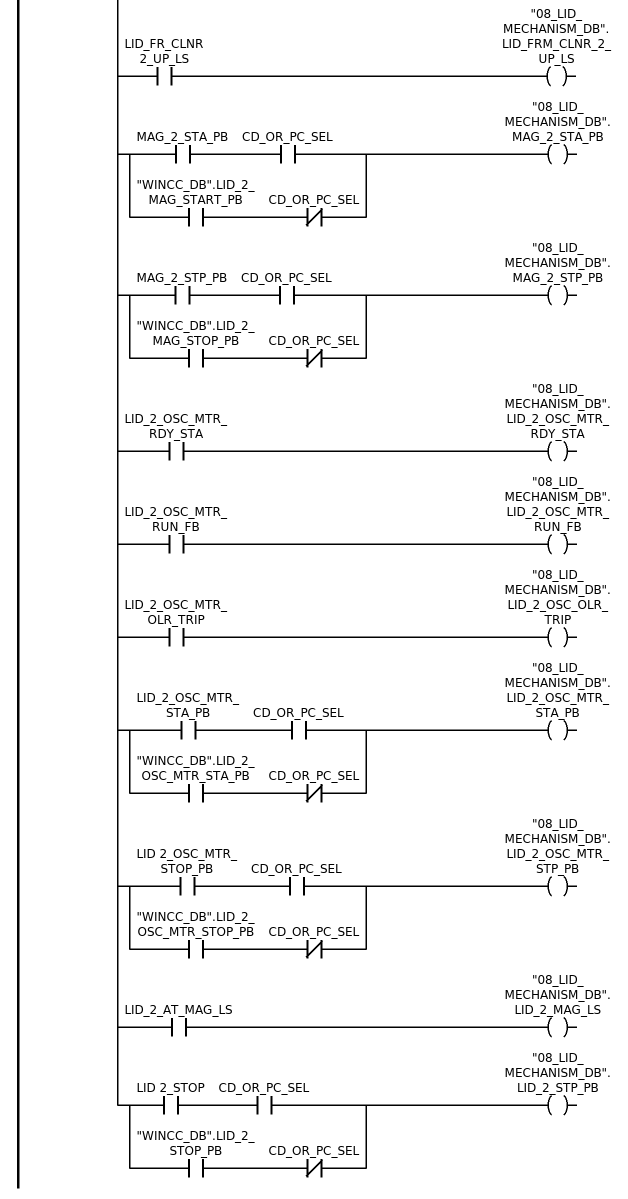
[picture p24: INPUT_MAPPING networks 7-7]
NETWORK
TITLE = LID MECHANISM 2 INPUT MAPPING
      A     "ALWAYS_ON";
      =     L 0.0;
      A     L 0.0;
      A     "LID_FR_CLN_MT_2_RDY_STA";
      =     "08_LID_MECHANISM_DB".LID_FR_CLN_MTR_2_RDY_STA;
      A     L 0.0;
      A     "LID_FR_CLN_MTR_2_RUN_FB";
      =     "08_LID_MECHANISM_DB".LID_FR_CLN_MTR_2_RUN_FB;
      A     L 0.0;
      A     "LID_FR_CLN_MTR_2_OLR";
      =     "08_LID_MECHANISM_DB".LID_FR_CLN_MTR_2_OLR_TRP;
      A     L 0.0;
      A(;
      A     "LID_FR_CL_MT_2_STA_PB";
      A     "CD_OR_PC_SEL";
      O;
      A     "WINCC_DB".LID_2_FRA_CLRMTR_STA_PB;
      AN    "CD_OR_PC_SEL";
      );
      =     "08_LID_MECHANISM_DB".LID_FR_CL_MTR_2_STA_PB;
      A     L 0.0;
      A(;
      A     "LID_FR_CLN_MTR_2_STP_PB";
      A     "CD_OR_PC_SEL";
      O;
      A     "WINCC_DB".LID_2_FRA_CLRMTR_STOP_PB;
      AN    "CD_OR_PC_SEL";
      );
      =     "08_LID_MECHANISM_DB".LID_FR_CL_MTR_2_STP_PB;
      A     L 0.0;
      A(;
      A     "LID_LIFT_2_CAR_FWD_STA";
      A     "CD_OR_PC_SEL";
      O;
      A     "WINCC_DB".LID_2_CARGE_FWD_STA_PB;
      AN    "CD_OR_PC_SEL";
      );
      =     "08_LID_MECHANISM_DB".LID_LIFT_2_CAR_FWD_STA;
      A     L 0.0;
      A(;
      A     "LID_LIFT_2_CAR_RET_STA";
      A     "CD_OR_PC_SEL";
      O;
      A     "WINCC_DB".LID_2_CARGE_REV_STA_PB;
      AN    "CD_OR_PC_SEL";
      );
      =     "08_LID_MECHANISM_DB".LID_LIFT_2_CAR_RET_STA;
      A     L 0.0;
      A(;
      A     "LID_LIFT_2_VER_DN_STA";
      A     "CD_OR_PC_SEL";
      O;
      A     "WINCC_DB".LID_2_VER_DN_STA_PB;
      AN    "CD_OR_PC_SEL";
      );
      =     "08_LID_MECHANISM_DB".LID_LIFT_2_VER_DN_STA;
      A     L 0.0;
      A(;
      A     "LID_LIFT_2_VER_UP_STA";
      A     "CD_OR_PC_SEL";
      O;
      A     "WINCC_DB".LID_2_VER_UP_STA_PB;
      AN    "CD_OR_PC_SEL";
      );
      =     "08_LID_MECHANISM_DB".LID_LIFT_2_VER_UP_STA;
      A     L 0.0;
      A(;
      A     "LID_FR_CLNR_2_DN_STA";
      A     "CD_OR_PC_SEL";
      O;
      A     "WINCC_DB".LID_2_FRA_CLR_DN_STA;
      AN    "CD_OR_PC_SEL";
      );
      =     "08_LID_MECHANISM_DB".LID_2_FRM_CLNR_DN_STA;
      A     L 0.0;
      A(;
      A     "LID_FR_CLNR_2_UP_STA";
      A     "CD_OR_PC_SEL";
      O;
      A     "WINCC_DB".LID_2_FRA_CLR_UP_STA;
      AN    "CD_OR_PC_SEL";
      );
      =     "08_LID_MECHANISM_DB".LID_2_FRM_CLNR_UP_STA;
      A     L 0.0;
      A(;
      A     "TELES_2_DOWN_STA";
      A     "CD_OR_PC_SEL";
      O;
      A     "WINCC_DB".LID_2_TELES_DN_STA;
      AN    "CD_OR_PC_SEL";
      );
      =     "08_LID_MECHANISM_DB".LID_2_TELES_DN_STA_PB;
      A     L 0.0;
      A(;
      A     "TELES_2_UP_STA";
      A     "CD_OR_PC_SEL";
      O;
      A     "WINCC_DB".LID_2_TELES_UP_STA;
      AN    "CD_OR_PC_SEL";
      );
      =     "08_LID_MECHANISM_DB".LID_2_TELES_UP_STA_PB;
      A     L 0.0;
      A     "LID_LIFT_2_CARR_FWD_LS";
      =     "08_LID_MECHANISM_DB".LID_LIFT_2_CAR_FWD_LS;
      A     L 0.0;
      A     "LID_LIFT_2_CARR_RET_LS";
      =     "08_LID_MECHANISM_DB".LID_LIFT_2_CAR_RET_LS;
      A     L 0.0;
      A     "LID_LIFT_2_VER_DN_LS";
      =     "08_LID_MECHANISM_DB".LID_LIFT_2_VER_DN_LS;
      A     L 0.0;
      A     "LID_LIFT_2_VER_UP_LS";
      =     "08_LID_MECHANISM_DB".LID_LIFT_2_VER_UP_LS;
      A     L 0.0;
      A     "TELES_2_DOWN_LS";
      =     "08_LID_MECHANISM_DB".TELE_2_DN_LS;
      A     L 0.0;
      A     "TELES_2_UP_LS";
      =     "08_LID_MECHANISM_DB".TELE_2_UP_LS;
      A     L 0.0;
      A     "LID_LIFT_2_CLN_POS_LS";
      =     "08_LID_MECHANISM_DB".LID_LIFT_2_CLN_LS;
      A     L 0.0;
      A     "LID_FR_CLNR_2_DOWN_LS";
      =     "08_LID_MECHANISM_DB".LID_FRM_CLNR_2_DN_LS;
      A     L 0.0;
      A     "LID_FR_CLNR 2_UP_LS";
      =     "08_LID_MECHANISM_DB".LID_FRM_CLNR_2_UP_LS;
      A     L 0.0;
      A(;
      A     "MAG_2_STA_PB";
      A     "CD_OR_PC_SEL";
      O;
      A     "WINCC_DB".LID_2_MAG_START_PB;
      AN    "CD_OR_PC_SEL";
      );
      =     "08_LID_MECHANISM_DB".MAG_2_STA_PB;
      A     L 0.0;
      A(;
      A     "MAG_2_STP_PB";
      A     "CD_OR_PC_SEL";
      O;
      A     "WINCC_DB".LID_2_MAG_STOP_PB;
      AN    "CD_OR_PC_SEL";
      );
      =     "08_LID_MECHANISM_DB".MAG_2_STP_PB;
      A     L 0.0;
      A     "LID_2_OSC_MTR_RDY_STA";
      =     "08_LID_MECHANISM_DB".LID_2_OSC_MTR_RDY_STA;
      A     L 0.0;
      A     "LID_2_OSC_MTR_RUN_FB";
      =     "08_LID_MECHANISM_DB".LID_2_OSC_MTR_RUN_FB;
      A     L 0.0;
      A     "LID_2_OSC_MTR_OLR_TRIP";
      =     "08_LID_MECHANISM_DB".LID_2_OSC_OLR_TRIP;
      A     L 0.0;
      A(;
      A     "LID_2_OSC_MTR_STA_PB";
      A     "CD_OR_PC_SEL";
      O;
      A     "WINCC_DB".LID_2_OSC_MTR_STA_PB;
      AN    "CD_OR_PC_SEL";
      );
      =     "08_LID_MECHANISM_DB".LID_2_OSC_MTR_STA_PB;
      A     L 0.0;
      A(;
      A     "LID 2_OSC_MTR_STOP_PB";
      A     "CD_OR_PC_SEL";
      O;
      A     "WINCC_DB".LID_2_OSC_MTR_STOP_PB;
      AN    "CD_OR_PC_SEL";
      );
      =     "08_LID_MECHANISM_DB".LID_2_OSC_MTR_STP_PB;
      A     L 0.0;
      A     "LID_2_AT_MAG_LS";
      =     "08_LID_MECHANISM_DB".LID_2_MAG_LS;
      A     L 0.0;
      A(;
      A     "LID 2_STOP";
      A     "CD_OR_PC_SEL";
      O;
      A     "WINCC_DB".LID_2_STOP_PB;
      AN    "CD_OR_PC_SEL";
      );
      =     "08_LID_MECHANISM_DB".LID_2_STP_PB;
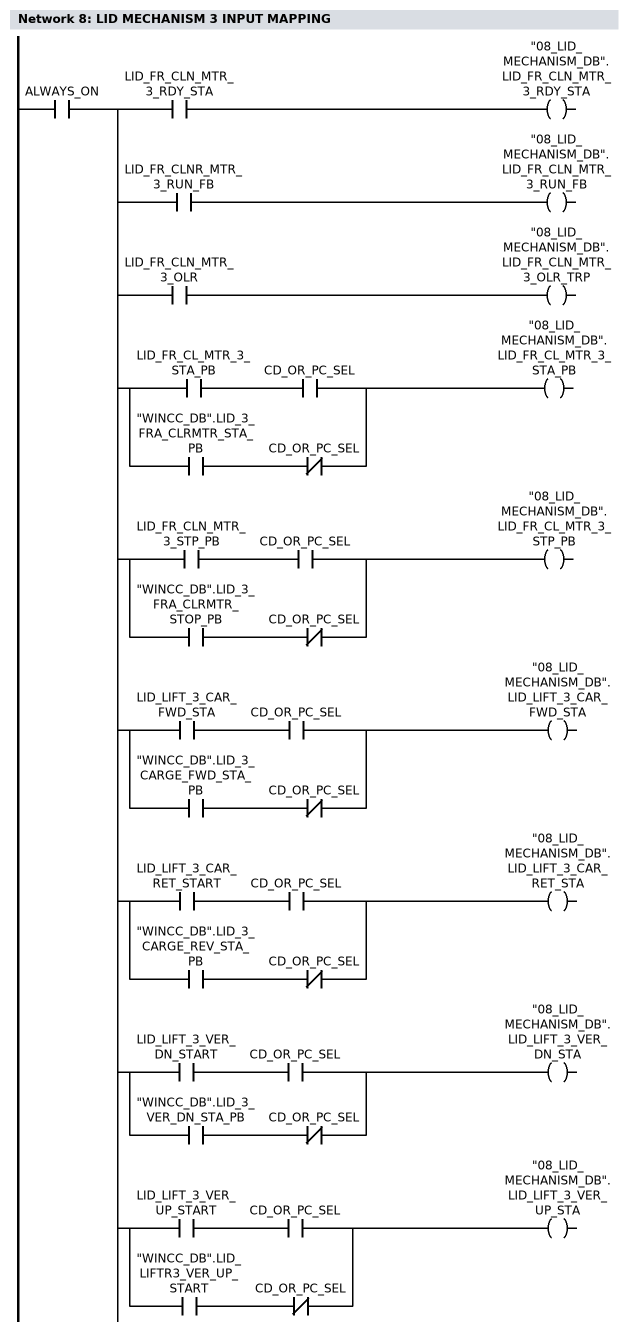
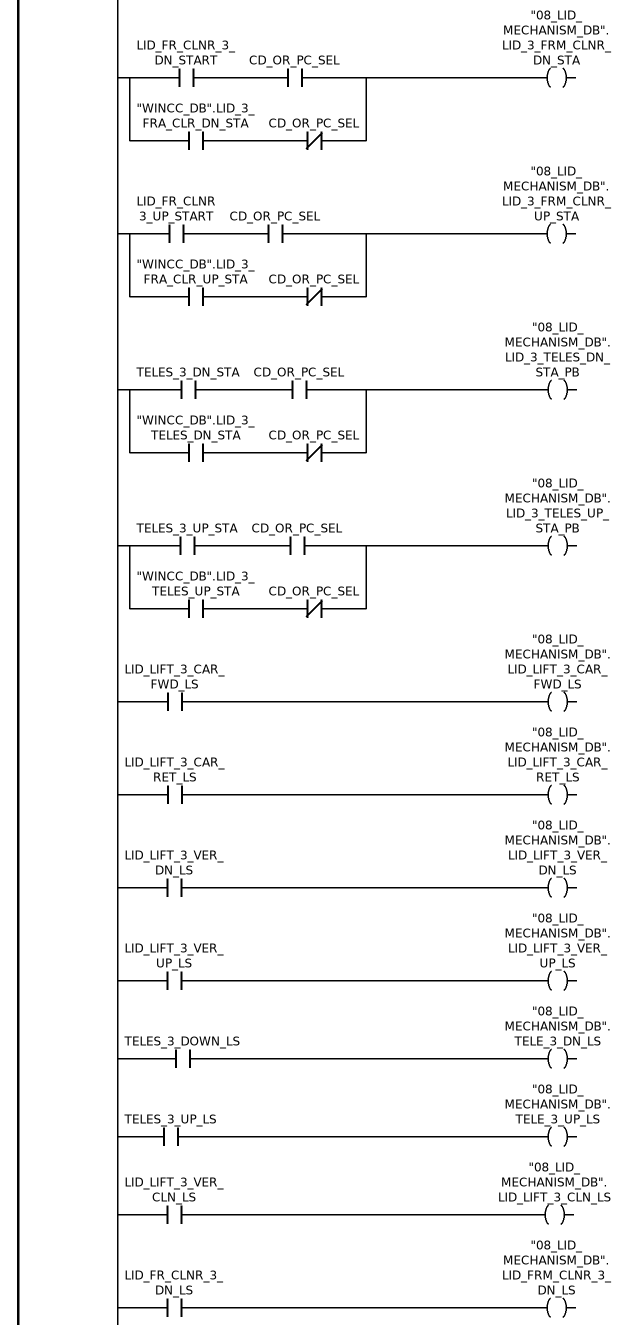
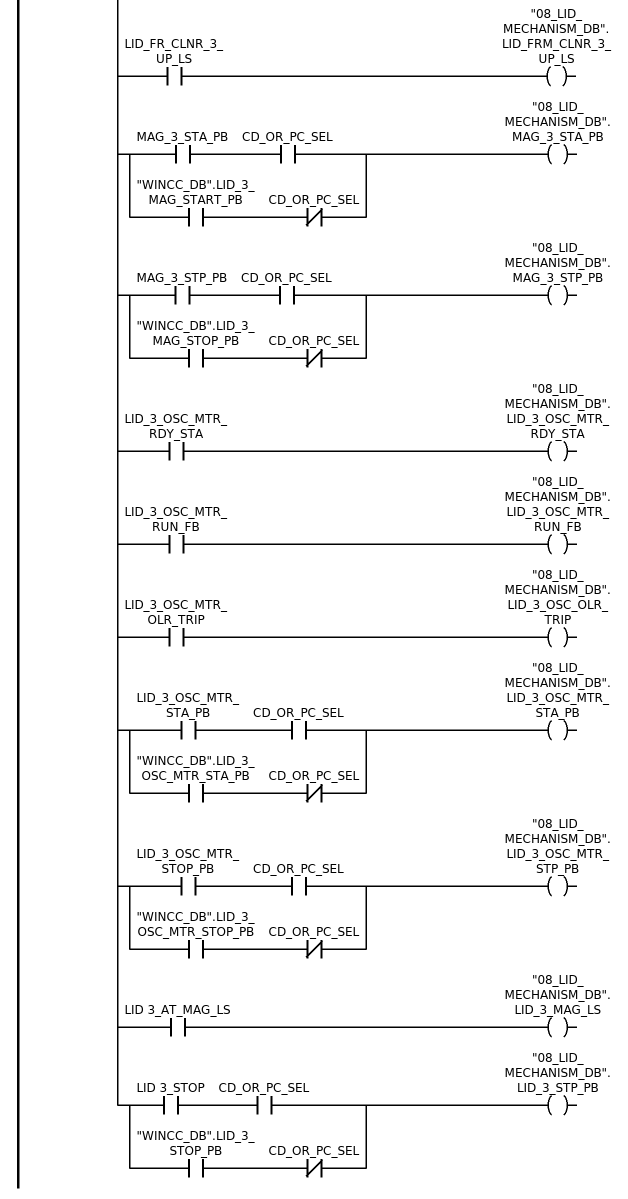
NETWORK
TITLE = LID MECHANISM 3 INPUT MAPPING
      A     "ALWAYS_ON";
      =     L 0.0;
      A     L 0.0;
      A     "LID_FR_CLN_MTR_3_RDY_STA";
      =     "08_LID_MECHANISM_DB".LID_FR_CLN_MTR_3_RDY_STA;
      A     L 0.0;
      A     "LID_FR_CLNR_MTR_3_RUN_FB";
      =     "08_LID_MECHANISM_DB".LID_FR_CLN_MTR_3_RUN_FB;
      A     L 0.0;
      A     "LID_FR_CLN_MTR_3_OLR";
      =     "08_LID_MECHANISM_DB".LID_FR_CLN_MTR_3_OLR_TRP;
      A     L 0.0;
      A(;
      A     "LID_FR_CL_MTR_3_STA_PB";
      A     "CD_OR_PC_SEL";
      O;
      A     "WINCC_DB".LID_3_FRA_CLRMTR_STA_PB;
      AN    "CD_OR_PC_SEL";
      );
      =     "08_LID_MECHANISM_DB".LID_FR_CL_MTR_3_STA_PB;
      A     L 0.0;
      A(;
      A     "LID_FR_CLN_MTR_3_STP_PB";
      A     "CD_OR_PC_SEL";
      O;
      A     "WINCC_DB".LID_3_FRA_CLRMTR_STOP_PB;
      AN    "CD_OR_PC_SEL";
      );
      =     "08_LID_MECHANISM_DB".LID_FR_CL_MTR_3_STP_PB;
      A     L 0.0;
      A(;
      A     "LID_LIFT_3_CAR_FWD_STA";
      A     "CD_OR_PC_SEL";
      O;
      A     "WINCC_DB".LID_3_CARGE_FWD_STA_PB;
      AN    "CD_OR_PC_SEL";
      );
      =     "08_LID_MECHANISM_DB".LID_LIFT_3_CAR_FWD_STA;
      A     L 0.0;
      A(;
      A     "LID_LIFT_3_CAR_RET_START";
      A     "CD_OR_PC_SEL";
      O;
      A     "WINCC_DB".LID_3_CARGE_REV_STA_PB;
      AN    "CD_OR_PC_SEL";
      );
      =     "08_LID_MECHANISM_DB".LID_LIFT_3_CAR_RET_STA;
      A     L 0.0;
      A(;
      A     "LID_LIFT_3_VER_DN_START";
      A     "CD_OR_PC_SEL";
      O;
      A     "WINCC_DB".LID_3_VER_DN_STA_PB;
      AN    "CD_OR_PC_SEL";
      );
      =     "08_LID_MECHANISM_DB".LID_LIFT_3_VER_DN_STA;
      A     L 0.0;
      A(;
      A     "LID_LIFT_3_VER_UP_START";
      A     "CD_OR_PC_SEL";
      O;
      A     "WINCC_DB".LID_LIFTR3_VER_UP_START;
      AN    "CD_OR_PC_SEL";
      );
      =     "08_LID_MECHANISM_DB".LID_LIFT_3_VER_UP_STA;
      A     L 0.0;
      A(;
      A     "LID_FR_CLNR_3_DN_START";
      A     "CD_OR_PC_SEL";
      O;
      A     "WINCC_DB".LID_3_FRA_CLR_DN_STA;
      AN    "CD_OR_PC_SEL";
      );
      =     "08_LID_MECHANISM_DB".LID_3_FRM_CLNR_DN_STA;
      A     L 0.0;
      A(;
      A     "LID_FR_CLNR 3_UP_START";
      A     "CD_OR_PC_SEL";
      O;
      A     "WINCC_DB".LID_3_FRA_CLR_UP_STA;
      AN    "CD_OR_PC_SEL";
      );
      =     "08_LID_MECHANISM_DB".LID_3_FRM_CLNR_UP_STA;
      A     L 0.0;
      A(;
      A     "TELES_3_DN_STA";
      A     "CD_OR_PC_SEL";
      O;
      A     "WINCC_DB".LID_3_TELES_DN_STA;
      AN    "CD_OR_PC_SEL";
      );
      =     "08_LID_MECHANISM_DB".LID_3_TELES_DN_STA_PB;
      A     L 0.0;
      A(;
      A     "TELES_3_UP_STA";
      A     "CD_OR_PC_SEL";
      O;
      A     "WINCC_DB".LID_3_TELES_UP_STA;
      AN    "CD_OR_PC_SEL";
      );
      =     "08_LID_MECHANISM_DB".LID_3_TELES_UP_STA_PB;
      A     L 0.0;
      A     "LID_LIFT_3_CAR_FWD_LS";
      =     "08_LID_MECHANISM_DB".LID_LIFT_3_CAR_FWD_LS;
      A     L 0.0;
      A     "LID_LIFT_3_CAR_RET_LS";
      =     "08_LID_MECHANISM_DB".LID_LIFT_3_CAR_RET_LS;
      A     L 0.0;
      A     "LID_LIFT_3_VER_DN_LS";
      =     "08_LID_MECHANISM_DB".LID_LIFT_3_VER_DN_LS;
      A     L 0.0;
      A     "LID_LIFT_3_VER_UP_LS";
      =     "08_LID_MECHANISM_DB".LID_LIFT_3_VER_UP_LS;
      A     L 0.0;
      A     "TELES_3_DOWN_LS";
      =     "08_LID_MECHANISM_DB".TELE_3_DN_LS;
      A     L 0.0;
      A     "TELES_3_UP_LS";
      =     "08_LID_MECHANISM_DB".TELE_3_UP_LS;
      A     L 0.0;
      A     "LID_LIFT_3_VER_CLN_LS";
      =     "08_LID_MECHANISM_DB".LID_LIFT_3_CLN_LS;
      A     L 0.0;
      A     "LID_FR_CLNR_3_DN_LS";
      =     "08_LID_MECHANISM_DB".LID_FRM_CLNR_3_DN_LS;
      A     L 0.0;
      A     "LID_FR_CLNR_3_UP_LS";
      =     "08_LID_MECHANISM_DB".LID_FRM_CLNR_3_UP_LS;
      A     L 0.0;
      A(;
      A     "MAG_3_STA_PB";
      A     "CD_OR_PC_SEL";
      O;
      A     "WINCC_DB".LID_3_MAG_START_PB;
      AN    "CD_OR_PC_SEL";
      );
      =     "08_LID_MECHANISM_DB".MAG_3_STA_PB;
      A     L 0.0;
      A(;
      A     "MAG_3_STP_PB";
      A     "CD_OR_PC_SEL";
      O;
      A     "WINCC_DB".LID_3_MAG_STOP_PB;
      AN    "CD_OR_PC_SEL";
      );
      =     "08_LID_MECHANISM_DB".MAG_3_STP_PB;
      A     L 0.0;
      A     "LID_3_OSC_MTR_RDY_STA";
      =     "08_LID_MECHANISM_DB".LID_3_OSC_MTR_RDY_STA;
      A     L 0.0;
      A     "LID_3_OSC_MTR_RUN_FB";
      =     "08_LID_MECHANISM_DB".LID_3_OSC_MTR_RUN_FB;
      A     L 0.0;
      A     "LID_3_OSC_MTR_OLR_TRIP";
      =     "08_LID_MECHANISM_DB".LID_3_OSC_OLR_TRIP;
      A     L 0.0;
      A(;
      A     "LID_3_OSC_MTR_STA_PB";
      A     "CD_OR_PC_SEL";
      O;
      A     "WINCC_DB".LID_3_OSC_MTR_STA_PB;
      AN    "CD_OR_PC_SEL";
      );
      =     "08_LID_MECHANISM_DB".LID_3_OSC_MTR_STA_PB;
      A     L 0.0;
      A(;
      A     "LID_3_OSC_MTR_STOP_PB";
      A     "CD_OR_PC_SEL";
      O;
      A     "WINCC_DB".LID_3_OSC_MTR_STOP_PB;
      AN    "CD_OR_PC_SEL";
      );
      =     "08_LID_MECHANISM_DB".LID_3_OSC_MTR_STP_PB;
      A     L 0.0;
      A     "LID 3_AT_MAG_LS";
      =     "08_LID_MECHANISM_DB".LID_3_MAG_LS;
      A     L 0.0;
      A(;
      A     "LID 3_STOP";
      A     "CD_OR_PC_SEL";
      O;
      A     "WINCC_DB".LID_3_STOP_PB;
      AN    "CD_OR_PC_SEL";
      );
      =     "08_LID_MECHANISM_DB".LID_3_STP_PB;
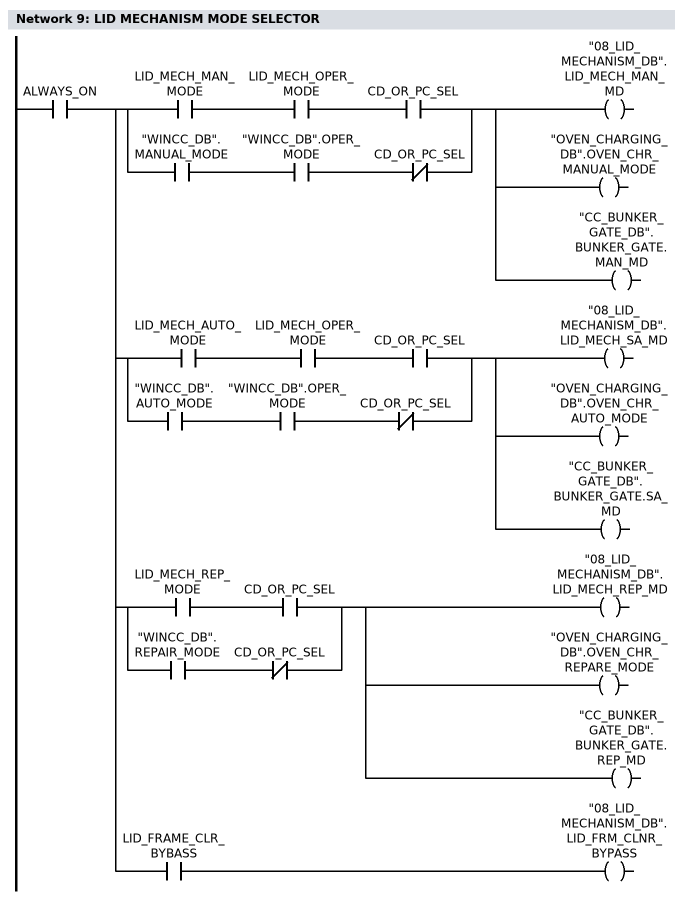
NETWORK
TITLE = LID MECHANISM MODE SELECTOR
      A     "ALWAYS_ON";
      =     L 0.0;
      A     L 0.0;
      A(;
      A     "LID_MECH_MAN_MODE";
      A     "LID_MECH_OPER_MODE";
      A     "CD_OR_PC_SEL";
      O;
      A     "WINCC_DB".MANUAL_MODE;
      A     "WINCC_DB".OPER_MODE;
      AN    "CD_OR_PC_SEL";
      );
      =     "08_LID_MECHANISM_DB".LID_MECH_MAN_MD;
      =     "OVEN_CHARGING_DB".OVEN_CHR_MANUAL_MODE;
      =     "CC_BUNKER_GATE_DB".BUNKER_GATE.MAN_MD;
      A     L 0.0;
      A(;
      A     "LID_MECH_AUTO_MODE";
      A     "LID_MECH_OPER_MODE";
      A     "CD_OR_PC_SEL";
      O;
      A     "WINCC_DB".AUTO_MODE;
      A     "WINCC_DB".OPER_MODE;
      AN    "CD_OR_PC_SEL";
      );
      =     "08_LID_MECHANISM_DB".LID_MECH_SA_MD;
      =     "OVEN_CHARGING_DB".OVEN_CHR_AUTO_MODE;
      =     "CC_BUNKER_GATE_DB".BUNKER_GATE.SA_MD;
      A     L 0.0;
      A(;
      A     "LID_MECH_REP_MODE";
      A     "CD_OR_PC_SEL";
      O;
      A     "WINCC_DB".REPAIR_MODE;
      AN    "CD_OR_PC_SEL";
      );
      =     "08_LID_MECHANISM_DB".LID_MECH_REP_MD;
      =     "OVEN_CHARGING_DB".OVEN_CHR_REPARE_MODE;
      =     "CC_BUNKER_GATE_DB".BUNKER_GATE.REP_MD;
      A     L 0.0;
      A     "LID_FRAME_CLR_BYBASS";
      =     "08_LID_MECHANISM_DB".LID_FRM_CLNR_BYPASS;
END_FUNCTION

FUNCTION "OUTPUT_MAPPING" : VOID	// FC 6
AUTHOR : Arun_Ram
VERSION : 0.1
BEGIN
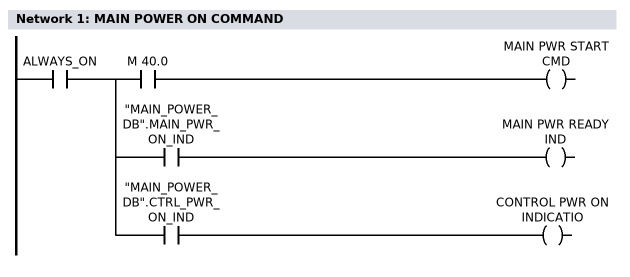
NETWORK
TITLE = MAIN POWER ON COMMAND
      A     "ALWAYS_ON";
      =     L 0.0;
      A     L 0.0;
      A     M 40.0;
      =     "MAIN PWR START CMD";
      A     L 0.0;
      A     "MAIN_POWER_DB".MAIN_PWR_ON_IND;
      =     "MAIN PWR READY IND";
      A     L 0.0;
      A     "MAIN_POWER_DB".CTRL_PWR_ON_IND;
      =     "CONTROL PWR ON INDICATIO";
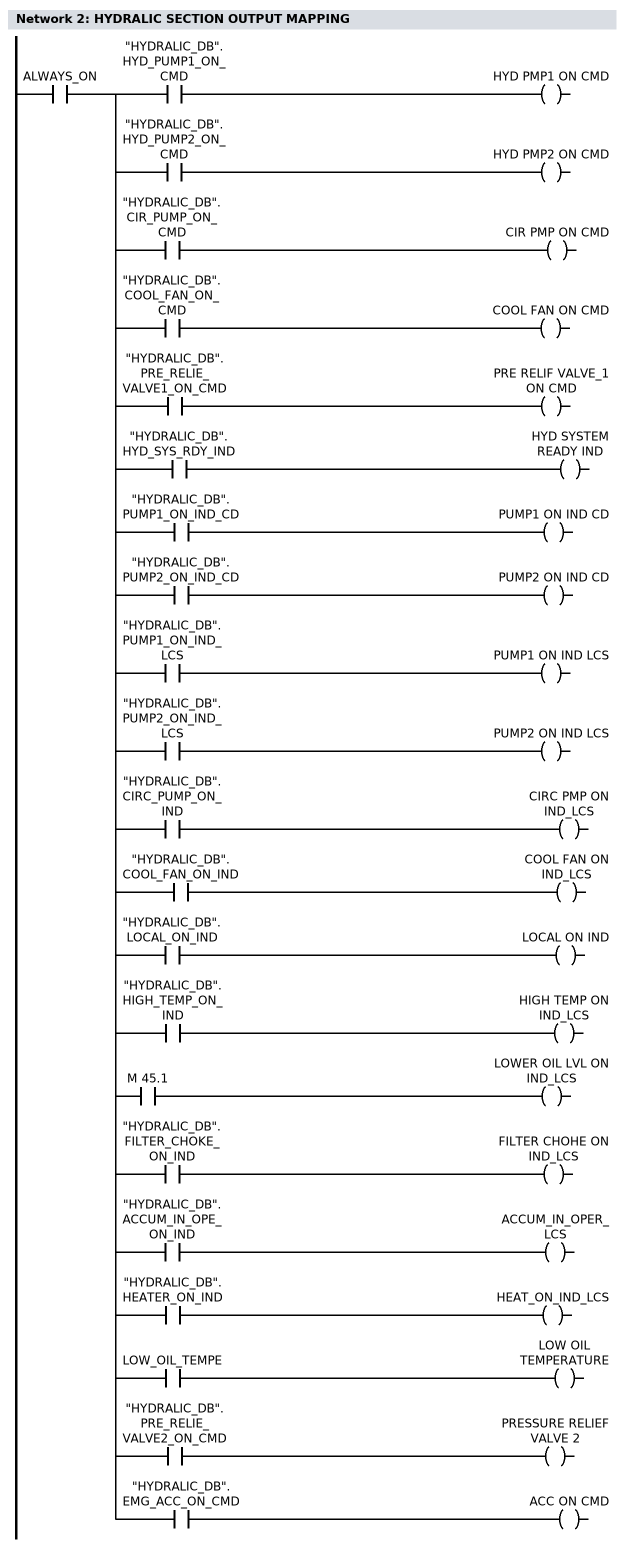
NETWORK
TITLE = HYDRALIC SECTION OUTPUT MAPPING
      A     "ALWAYS_ON";
      =     L 0.0;
      A     L 0.0;
      A     "HYDRALIC_DB".HYD_PUMP1_ON_CMD;
      =     "HYD PMP1 ON CMD";
      A     L 0.0;
      A     "HYDRALIC_DB".HYD_PUMP2_ON_CMD;
      =     "HYD PMP2 ON CMD";
      A     L 0.0;
      A     "HYDRALIC_DB".CIR_PUMP_ON_CMD;
      =     "CIR PMP ON CMD";
      A     L 0.0;
      A     "HYDRALIC_DB".COOL_FAN_ON_CMD;
      =     "COOL FAN ON CMD";
      A     L 0.0;
      A     "HYDRALIC_DB".PRE_RELIE_VALVE1_ON_CMD;
      =     "PRE RELIF VALVE_1 ON CMD";
      A     L 0.0;
      A     "HYDRALIC_DB".HYD_SYS_RDY_IND;
      =     "HYD SYSTEM READY IND";
      A     L 0.0;
      A     "HYDRALIC_DB".PUMP1_ON_IND_CD;
      =     "PUMP1 ON IND CD";
      A     L 0.0;
      A     "HYDRALIC_DB".PUMP2_ON_IND_CD;
      =     "PUMP2 ON IND CD";
      A     L 0.0;
      A     "HYDRALIC_DB".PUMP1_ON_IND_LCS;
      =     "PUMP1 ON IND LCS";
      A     L 0.0;
      A     "HYDRALIC_DB".PUMP2_ON_IND_LCS;
      =     "PUMP2 ON IND LCS";
      A     L 0.0;
      A     "HYDRALIC_DB".CIRC_PUMP_ON_IND;
      =     "CIRC PMP ON IND_LCS";
      A     L 0.0;
      A     "HYDRALIC_DB".COOL_FAN_ON_IND;
      =     "COOL FAN ON IND_LCS";
      A     L 0.0;
      A     "HYDRALIC_DB".LOCAL_ON_IND;
      =     "LOCAL ON IND";
      A     L 0.0;
      A     "HYDRALIC_DB".HIGH_TEMP_ON_IND;
      =     "HIGH TEMP ON IND_LCS";
      A     L 0.0;
      A     M 45.1;
      =     "LOWER OIL LVL ON IND_LCS";
      A     L 0.0;
      A     "HYDRALIC_DB".FILTER_CHOKE_ON_IND;
      =     "FILTER CHOHE ON IND_LCS";
      A     L 0.0;
      A     "HYDRALIC_DB".ACCUM_IN_OPE_ON_IND;
      =     "ACCUM_IN_OPER_LCS";
      A     L 0.0;
      A     "HYDRALIC_DB".HEATER_ON_IND;
      =     "HEAT_ON_IND_LCS";
      A     L 0.0;
      A     "LOW_OIL_TEMPE";
      =     "LOW OIL TEMPERATURE";
      A     L 0.0;
      A     "HYDRALIC_DB".PRE_RELIE_VALVE2_ON_CMD;
      =     "PRESSURE RELIEF VALVE 2";
      A     L 0.0;
      A     "HYDRALIC_DB".EMG_ACC_ON_CMD;
      =     "ACC ON CMD";
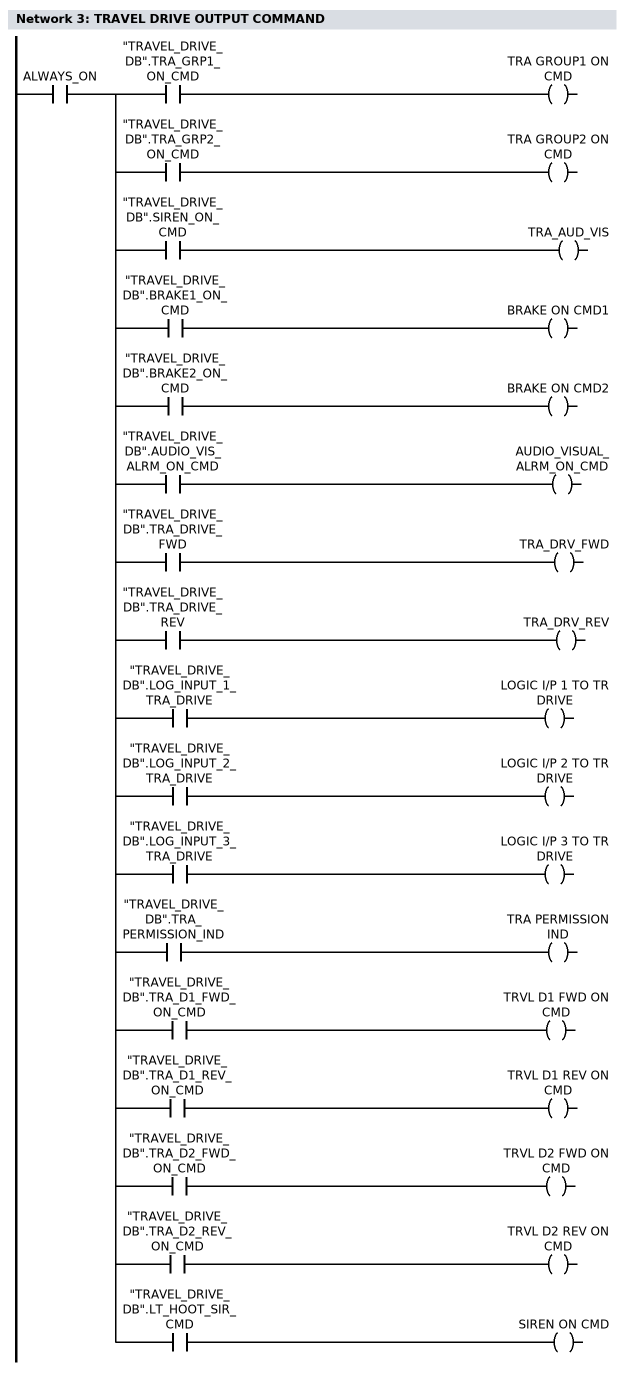
NETWORK
TITLE = TRAVEL DRIVE OUTPUT COMMAND
      A     "ALWAYS_ON";
      =     L 0.0;
      A     L 0.0;
      A     "TRAVEL_DRIVE_DB".TRA_GRP1_ON_CMD;
      =     "TRA GROUP1 ON CMD";
      A     L 0.0;
      A     "TRAVEL_DRIVE_DB".TRA_GRP2_ON_CMD;
      =     "TRA GROUP2 ON CMD";
      A     L 0.0;
      A     "TRAVEL_DRIVE_DB".SIREN_ON_CMD;
      =     "TRA_AUD_VIS";
      A     L 0.0;
      A     "TRAVEL_DRIVE_DB".BRAKE1_ON_CMD;
      =     "BRAKE ON CMD1";
      A     L 0.0;
      A     "TRAVEL_DRIVE_DB".BRAKE2_ON_CMD;
      =     "BRAKE ON CMD2";
      A     L 0.0;
      A     "TRAVEL_DRIVE_DB".AUDIO_VIS_ALRM_ON_CMD;
      =     "AUDIO_VISUAL_ALRM_ON_CMD";
      A     L 0.0;
      A     "TRAVEL_DRIVE_DB".TRA_DRIVE_FWD;
      =     "TRA_DRV_FWD";
      A     L 0.0;
      A     "TRAVEL_DRIVE_DB".TRA_DRIVE_REV;
      =     "TRA_DRV_REV";
      A     L 0.0;
      A     "TRAVEL_DRIVE_DB".LOG_INPUT_1_TRA_DRIVE;
      =     "LOGIC I/P 1 TO TR DRIVE";
      A     L 0.0;
      A     "TRAVEL_DRIVE_DB".LOG_INPUT_2_TRA_DRIVE;
      =     "LOGIC I/P 2 TO TR DRIVE";
      A     L 0.0;
      A     "TRAVEL_DRIVE_DB".LOG_INPUT_3_TRA_DRIVE;
      =     "LOGIC I/P 3 TO TR DRIVE";
      A     L 0.0;
      A     "TRAVEL_DRIVE_DB".TRA_PERMISSION_IND;
      =     "TRA PERMISSION IND";
      A     L 0.0;
      A     "TRAVEL_DRIVE_DB".TRA_D1_FWD_ON_CMD;
      =     "TRVL D1 FWD ON CMD";
      A     L 0.0;
      A     "TRAVEL_DRIVE_DB".TRA_D1_REV_ON_CMD;
      =     "TRVL D1 REV ON CMD";
      A     L 0.0;
      A     "TRAVEL_DRIVE_DB".TRA_D2_FWD_ON_CMD;
      =     "TRVL D2 FWD ON CMD";
      A     L 0.0;
      A     "TRAVEL_DRIVE_DB".TRA_D2_REV_ON_CMD;
      =     "TRVL D2 REV ON CMD";
      A     L 0.0;
      A     "TRAVEL_DRIVE_DB".LT_HOOT_SIR_CMD;
      =     "SIREN ON CMD";
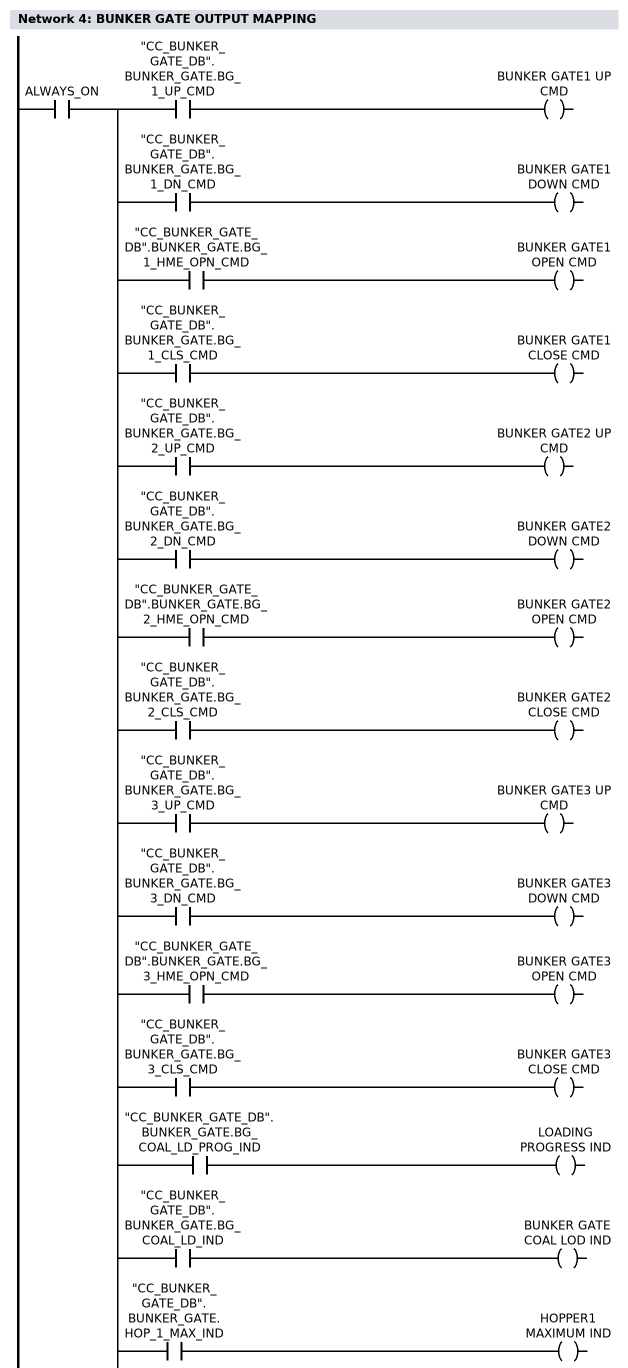
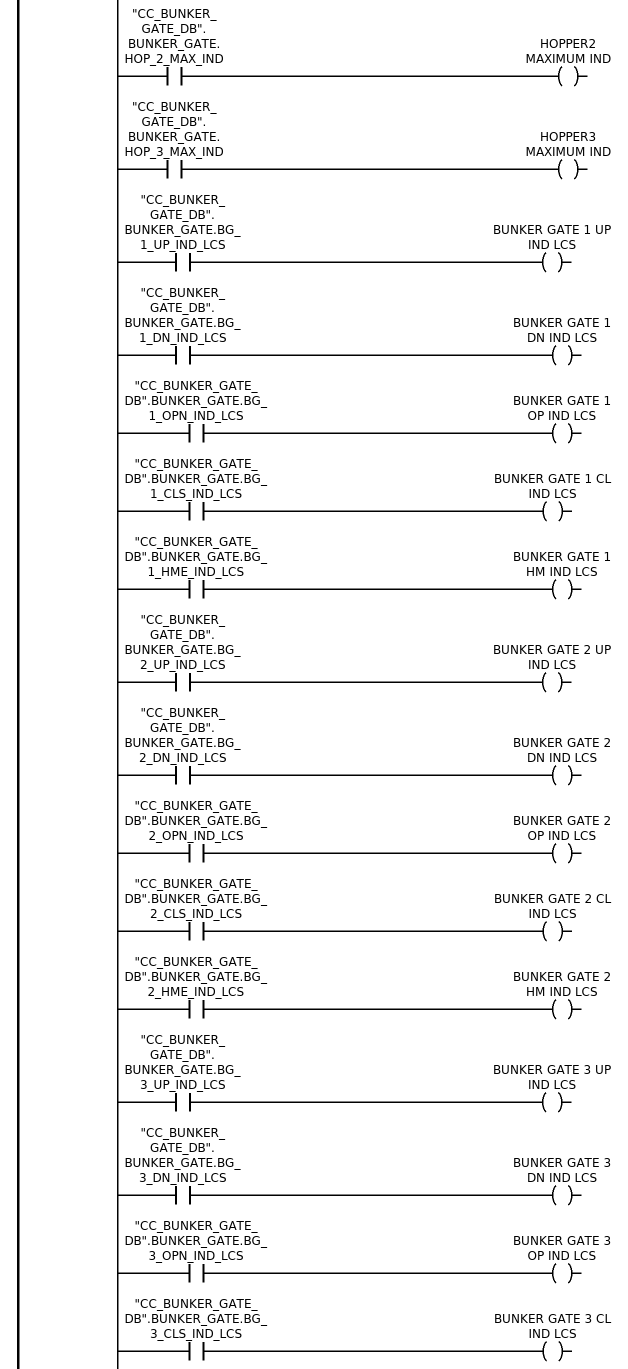
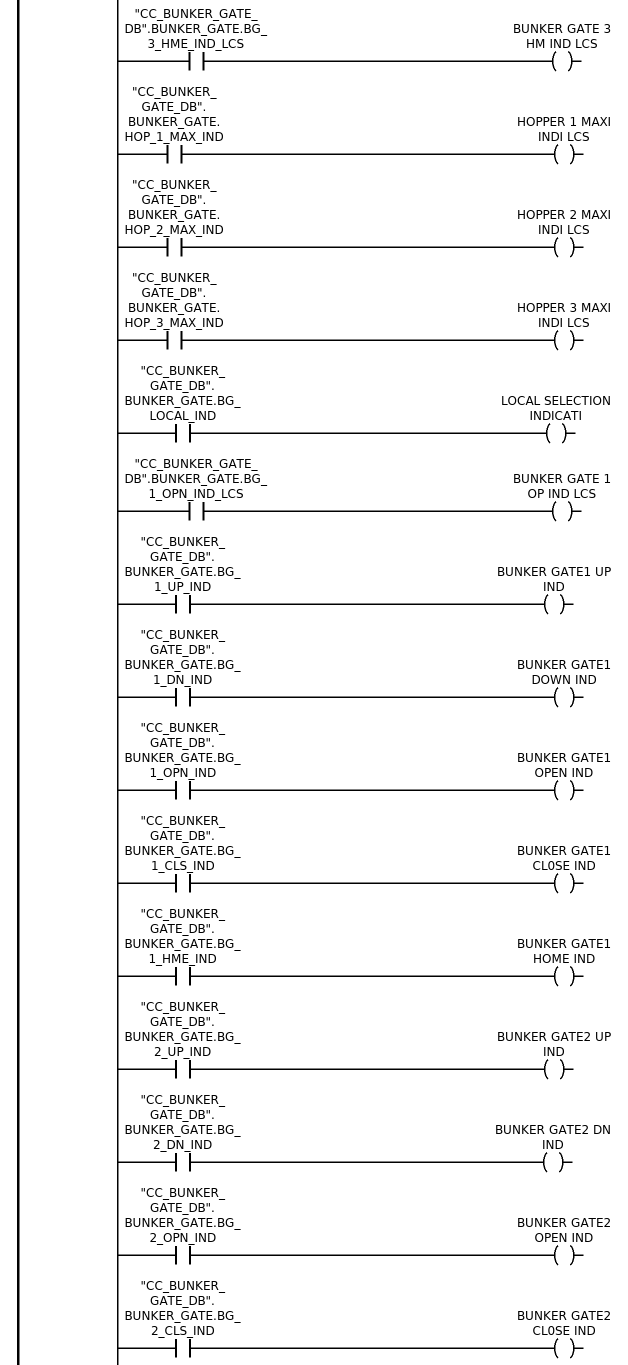
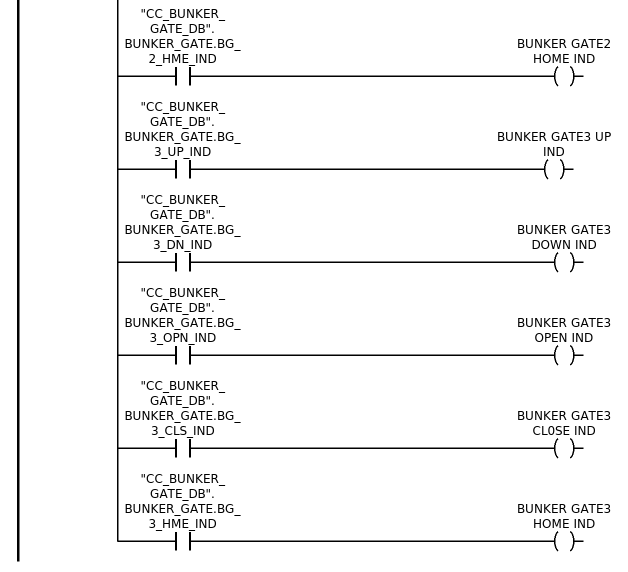
NETWORK
TITLE = BUNKER GATE OUTPUT MAPPING
      A     "ALWAYS_ON";
      =     L 0.0;
      A     L 0.0;
      A     "CC_BUNKER_GATE_DB".BUNKER_GATE.BG_1_UP_CMD;
      =     "BUNKER GATE1 UP CMD";
      A     L 0.0;
      A     "CC_BUNKER_GATE_DB".BUNKER_GATE.BG_1_DN_CMD;
      =     "BUNKER GATE1 DOWN CMD";
      A     L 0.0;
      A     "CC_BUNKER_GATE_DB".BUNKER_GATE.BG_1_HME_OPN_CMD;
      =     "BUNKER GATE1 OPEN CMD";
      A     L 0.0;
      A     "CC_BUNKER_GATE_DB".BUNKER_GATE.BG_1_CLS_CMD;
      =     "BUNKER GATE1 CLOSE CMD";
      A     L 0.0;
      A     "CC_BUNKER_GATE_DB".BUNKER_GATE.BG_2_UP_CMD;
      =     "BUNKER GATE2 UP CMD";
      A     L 0.0;
      A     "CC_BUNKER_GATE_DB".BUNKER_GATE.BG_2_DN_CMD;
      =     "BUNKER GATE2 DOWN CMD";
      A     L 0.0;
      A     "CC_BUNKER_GATE_DB".BUNKER_GATE.BG_2_HME_OPN_CMD;
      =     "BUNKER GATE2 OPEN CMD";
      A     L 0.0;
      A     "CC_BUNKER_GATE_DB".BUNKER_GATE.BG_2_CLS_CMD;
      =     "BUNKER GATE2 CLOSE CMD";
      A     L 0.0;
      A     "CC_BUNKER_GATE_DB".BUNKER_GATE.BG_3_UP_CMD;
      =     "BUNKER GATE3 UP CMD";
      A     L 0.0;
      A     "CC_BUNKER_GATE_DB".BUNKER_GATE.BG_3_DN_CMD;
      =     "BUNKER GATE3 DOWN CMD";
      A     L 0.0;
      A     "CC_BUNKER_GATE_DB".BUNKER_GATE.BG_3_HME_OPN_CMD;
      =     "BUNKER GATE3 OPEN CMD";
      A     L 0.0;
      A     "CC_BUNKER_GATE_DB".BUNKER_GATE.BG_3_CLS_CMD;
      =     "BUNKER GATE3 CLOSE CMD";
      A     L 0.0;
      A     "CC_BUNKER_GATE_DB".BUNKER_GATE.BG_COAL_LD_PROG_IND;
      =     "LOADING PROGRESS IND";
      A     L 0.0;
      A     "CC_BUNKER_GATE_DB".BUNKER_GATE.BG_COAL_LD_IND;
      =     "BUNKER GATE COAL LOD IND";
      A     L 0.0;
      A     "CC_BUNKER_GATE_DB".BUNKER_GATE.HOP_1_MAX_IND;
      =     "HOPPER1 MAXIMUM IND";
      A     L 0.0;
      A     "CC_BUNKER_GATE_DB".BUNKER_GATE.HOP_2_MAX_IND;
      =     "HOPPER2 MAXIMUM IND";
      A     L 0.0;
      A     "CC_BUNKER_GATE_DB".BUNKER_GATE.HOP_3_MAX_IND;
      =     "HOPPER3 MAXIMUM IND";
      A     L 0.0;
      A     "CC_BUNKER_GATE_DB".BUNKER_GATE.BG_1_UP_IND_LCS;
      =     "BUNKER GATE 1 UP IND LCS";
      A     L 0.0;
      A     "CC_BUNKER_GATE_DB".BUNKER_GATE.BG_1_DN_IND_LCS;
      =     "BUNKER GATE 1 DN IND LCS";
      A     L 0.0;
      A     "CC_BUNKER_GATE_DB".BUNKER_GATE.BG_1_OPN_IND_LCS;
      =     "BUNKER GATE 1 OP IND LCS";
      A     L 0.0;
      A     "CC_BUNKER_GATE_DB".BUNKER_GATE.BG_1_CLS_IND_LCS;
      =     "BUNKER GATE 1 CL IND LCS";
      A     L 0.0;
      A     "CC_BUNKER_GATE_DB".BUNKER_GATE.BG_1_HME_IND_LCS;
      =     "BUNKER GATE 1 HM IND LCS";
      A     L 0.0;
      A     "CC_BUNKER_GATE_DB".BUNKER_GATE.BG_2_UP_IND_LCS;
      =     "BUNKER GATE 2 UP IND LCS";
      A     L 0.0;
      A     "CC_BUNKER_GATE_DB".BUNKER_GATE.BG_2_DN_IND_LCS;
      =     "BUNKER GATE 2 DN IND LCS";
      A     L 0.0;
      A     "CC_BUNKER_GATE_DB".BUNKER_GATE.BG_2_OPN_IND_LCS;
      =     "BUNKER GATE 2 OP IND LCS";
      A     L 0.0;
      A     "CC_BUNKER_GATE_DB".BUNKER_GATE.BG_2_CLS_IND_LCS;
      =     "BUNKER GATE 2 CL IND LCS";
      A     L 0.0;
      A     "CC_BUNKER_GATE_DB".BUNKER_GATE.BG_2_HME_IND_LCS;
      =     "BUNKER GATE 2 HM IND LCS";
      A     L 0.0;
      A     "CC_BUNKER_GATE_DB".BUNKER_GATE.BG_3_UP_IND_LCS;
      =     "BUNKER GATE 3 UP IND LCS";
      A     L 0.0;
      A     "CC_BUNKER_GATE_DB".BUNKER_GATE.BG_3_DN_IND_LCS;
      =     "BUNKER GATE 3 DN IND LCS";
      A     L 0.0;
      A     "CC_BUNKER_GATE_DB".BUNKER_GATE.BG_3_OPN_IND_LCS;
      =     "BUNKER GATE 3 OP IND LCS";
      A     L 0.0;
      A     "CC_BUNKER_GATE_DB".BUNKER_GATE.BG_3_CLS_IND_LCS;
      =     "BUNKER GATE 3 CL IND LCS";
      A     L 0.0;
      A     "CC_BUNKER_GATE_DB".BUNKER_GATE.BG_3_HME_IND_LCS;
      =     "BUNKER GATE 3 HM IND LCS";
      A     L 0.0;
      A     "CC_BUNKER_GATE_DB".BUNKER_GATE.HOP_1_MAX_IND;
      =     "HOPPER 1 MAXI INDI LCS";
      A     L 0.0;
      A     "CC_BUNKER_GATE_DB".BUNKER_GATE.HOP_2_MAX_IND;
      =     "HOPPER 2 MAXI INDI LCS";
      A     L 0.0;
      A     "CC_BUNKER_GATE_DB".BUNKER_GATE.HOP_3_MAX_IND;
      =     "HOPPER 3 MAXI INDI LCS";
      A     L 0.0;
      A     "CC_BUNKER_GATE_DB".BUNKER_GATE.BG_LOCAL_IND;
      =     "LOCAL SELECTION INDICATI";
      A     L 0.0;
      A     "CC_BUNKER_GATE_DB".BUNKER_GATE.BG_1_OPN_IND_LCS;
      =     "BUNKER GATE 1 OP IND LCS";
      A     L 0.0;
      A     "CC_BUNKER_GATE_DB".BUNKER_GATE.BG_1_UP_IND;
      =     "BUNKER GATE1 UP IND";
      A     L 0.0;
      A     "CC_BUNKER_GATE_DB".BUNKER_GATE.BG_1_DN_IND;
      =     "BUNKER GATE1 DOWN IND";
      A     L 0.0;
      A     "CC_BUNKER_GATE_DB".BUNKER_GATE.BG_1_OPN_IND;
      =     "BUNKER GATE1 OPEN IND";
      A     L 0.0;
      A     "CC_BUNKER_GATE_DB".BUNKER_GATE.BG_1_CLS_IND;
      =     "BUNKER GATE1 CL0SE IND";
      A     L 0.0;
      A     "CC_BUNKER_GATE_DB".BUNKER_GATE.BG_1_HME_IND;
      =     "BUNKER GATE1 HOME IND";
      A     L 0.0;
      A     "CC_BUNKER_GATE_DB".BUNKER_GATE.BG_2_UP_IND;
      =     "BUNKER GATE2 UP IND";
      A     L 0.0;
      A     "CC_BUNKER_GATE_DB".BUNKER_GATE.BG_2_DN_IND;
      =     "BUNKER GATE2 DN IND";
      A     L 0.0;
      A     "CC_BUNKER_GATE_DB".BUNKER_GATE.BG_2_OPN_IND;
      =     "BUNKER GATE2 OPEN IND";
      A     L 0.0;
      A     "CC_BUNKER_GATE_DB".BUNKER_GATE.BG_2_CLS_IND;
      =     "BUNKER GATE2 CL0SE IND";
      A     L 0.0;
      A     "CC_BUNKER_GATE_DB".BUNKER_GATE.BG_2_HME_IND;
      =     "BUNKER GATE2 HOME IND";
      A     L 0.0;
      A     "CC_BUNKER_GATE_DB".BUNKER_GATE.BG_3_UP_IND;
      =     "BUNKER GATE3 UP IND";
      A     L 0.0;
      A     "CC_BUNKER_GATE_DB".BUNKER_GATE.BG_3_DN_IND;
      =     "BUNKER GATE3 DOWN IND";
      A     L 0.0;
      A     "CC_BUNKER_GATE_DB".BUNKER_GATE.BG_3_OPN_IND;
      =     "BUNKER GATE3 OPEN IND";
      A     L 0.0;
      A     "CC_BUNKER_GATE_DB".BUNKER_GATE.BG_3_CLS_IND;
      =     "BUNKER GATE3 CL0SE IND";
      A     L 0.0;
      A     "CC_BUNKER_GATE_DB".BUNKER_GATE.BG_3_HME_IND;
      =     "BUNKER GATE3 HOME IND";
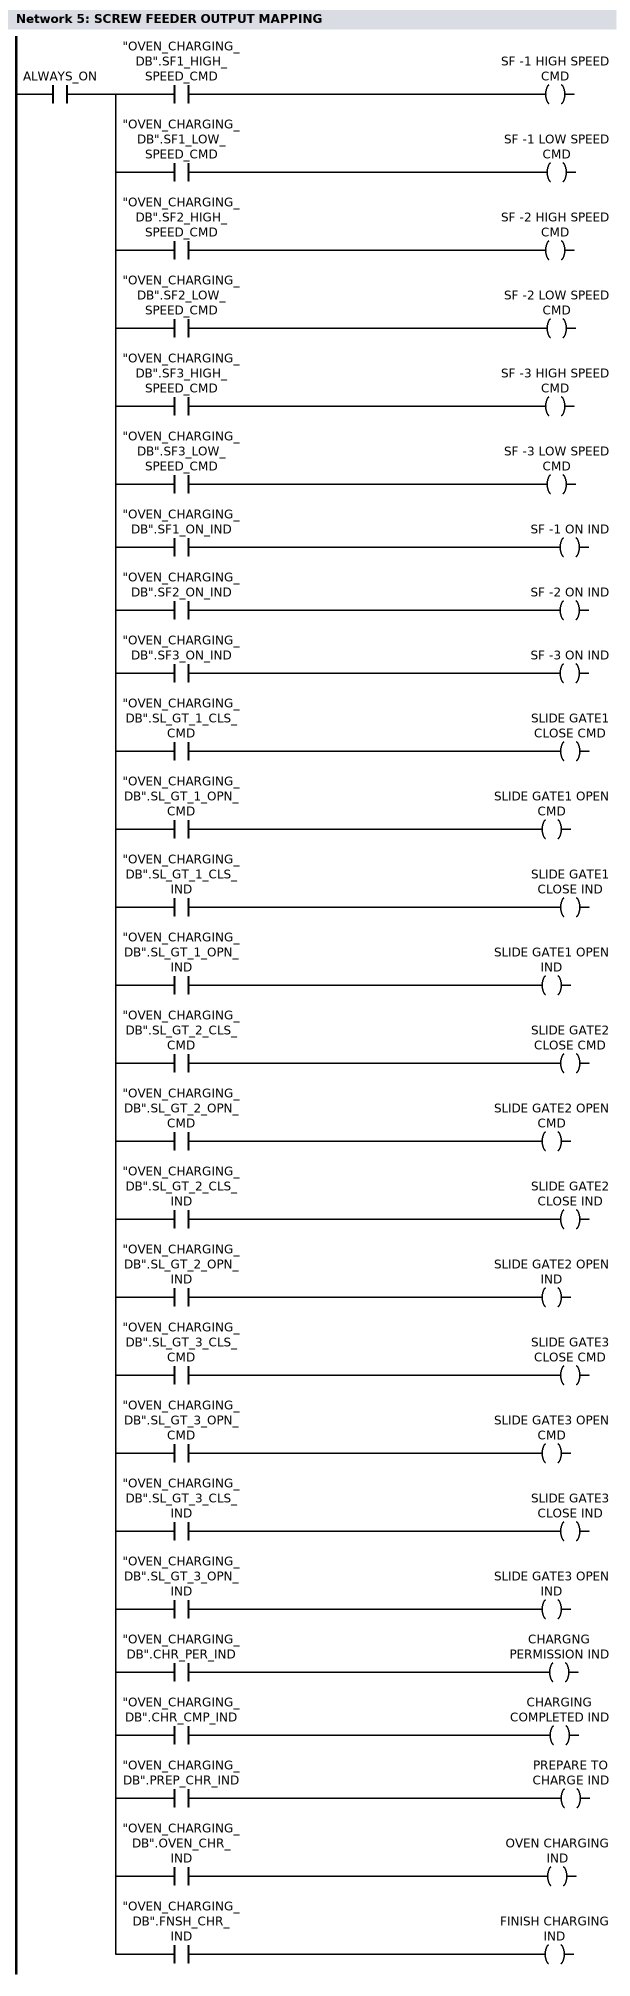
NETWORK
TITLE = SCREW FEEDER OUTPUT MAPPING
      A     "ALWAYS_ON";
      =     L 0.0;
      A     L 0.0;
      A     "OVEN_CHARGING_DB".SF1_HIGH_SPEED_CMD;
      =     "SF -1 HIGH SPEED CMD";
      A     L 0.0;
      A     "OVEN_CHARGING_DB".SF1_LOW_SPEED_CMD;
      =     "SF -1 LOW SPEED CMD";
      A     L 0.0;
      A     "OVEN_CHARGING_DB".SF2_HIGH_SPEED_CMD;
      =     "SF -2 HIGH SPEED CMD";
      A     L 0.0;
      A     "OVEN_CHARGING_DB".SF2_LOW_SPEED_CMD;
      =     "SF -2 LOW SPEED CMD";
      A     L 0.0;
      A     "OVEN_CHARGING_DB".SF3_HIGH_SPEED_CMD;
      =     "SF -3 HIGH SPEED CMD";
      A     L 0.0;
      A     "OVEN_CHARGING_DB".SF3_LOW_SPEED_CMD;
      =     "SF -3 LOW SPEED CMD";
      A     L 0.0;
      A     "OVEN_CHARGING_DB".SF1_ON_IND;
      =     "SF -1 ON IND";
      A     L 0.0;
      A     "OVEN_CHARGING_DB".SF2_ON_IND;
      =     "SF -2 ON IND";
      A     L 0.0;
      A     "OVEN_CHARGING_DB".SF3_ON_IND;
      =     "SF -3 ON IND";
      A     L 0.0;
      A     "OVEN_CHARGING_DB".SL_GT_1_CLS_CMD;
      =     "SLIDE GATE1 CLOSE CMD";
      A     L 0.0;
      A     "OVEN_CHARGING_DB".SL_GT_1_OPN_CMD;
      =     "SLIDE GATE1 OPEN CMD";
      A     L 0.0;
      A     "OVEN_CHARGING_DB".SL_GT_1_CLS_IND;
      =     "SLIDE GATE1 CLOSE IND";
      A     L 0.0;
      A     "OVEN_CHARGING_DB".SL_GT_1_OPN_IND;
      =     "SLIDE GATE1 OPEN IND";
      A     L 0.0;
      A     "OVEN_CHARGING_DB".SL_GT_2_CLS_CMD;
      =     "SLIDE GATE2 CLOSE CMD";
      A     L 0.0;
      A     "OVEN_CHARGING_DB".SL_GT_2_OPN_CMD;
      =     "SLIDE GATE2 OPEN CMD";
      A     L 0.0;
      A     "OVEN_CHARGING_DB".SL_GT_2_CLS_IND;
      =     "SLIDE GATE2 CLOSE IND";
      A     L 0.0;
      A     "OVEN_CHARGING_DB".SL_GT_2_OPN_IND;
      =     "SLIDE GATE2 OPEN IND";
      A     L 0.0;
      A     "OVEN_CHARGING_DB".SL_GT_3_CLS_CMD;
      =     "SLIDE GATE3 CLOSE CMD";
      A     L 0.0;
      A     "OVEN_CHARGING_DB".SL_GT_3_OPN_CMD;
      =     "SLIDE GATE3 OPEN CMD";
      A     L 0.0;
      A     "OVEN_CHARGING_DB".SL_GT_3_CLS_IND;
      =     "SLIDE GATE3 CLOSE IND";
      A     L 0.0;
      A     "OVEN_CHARGING_DB".SL_GT_3_OPN_IND;
      =     "SLIDE GATE3 OPEN IND";
      A     L 0.0;
      A     "OVEN_CHARGING_DB".CHR_PER_IND;
      =     "CHARGNG PERMISSION IND";
      A     L 0.0;
      A     "OVEN_CHARGING_DB".CHR_CMP_IND;
      =     "CHARGING COMPLETED IND";
      A     L 0.0;
      A     "OVEN_CHARGING_DB".PREP_CHR_IND;
      =     "PREPARE TO CHARGE IND";
      A     L 0.0;
      A     "OVEN_CHARGING_DB".OVEN_CHR_IND;
      =     "OVEN CHARGING IND";
      A     L 0.0;
      A     "OVEN_CHARGING_DB".FNSH_CHR_IND;
      =     "FINISH CHARGING IND";
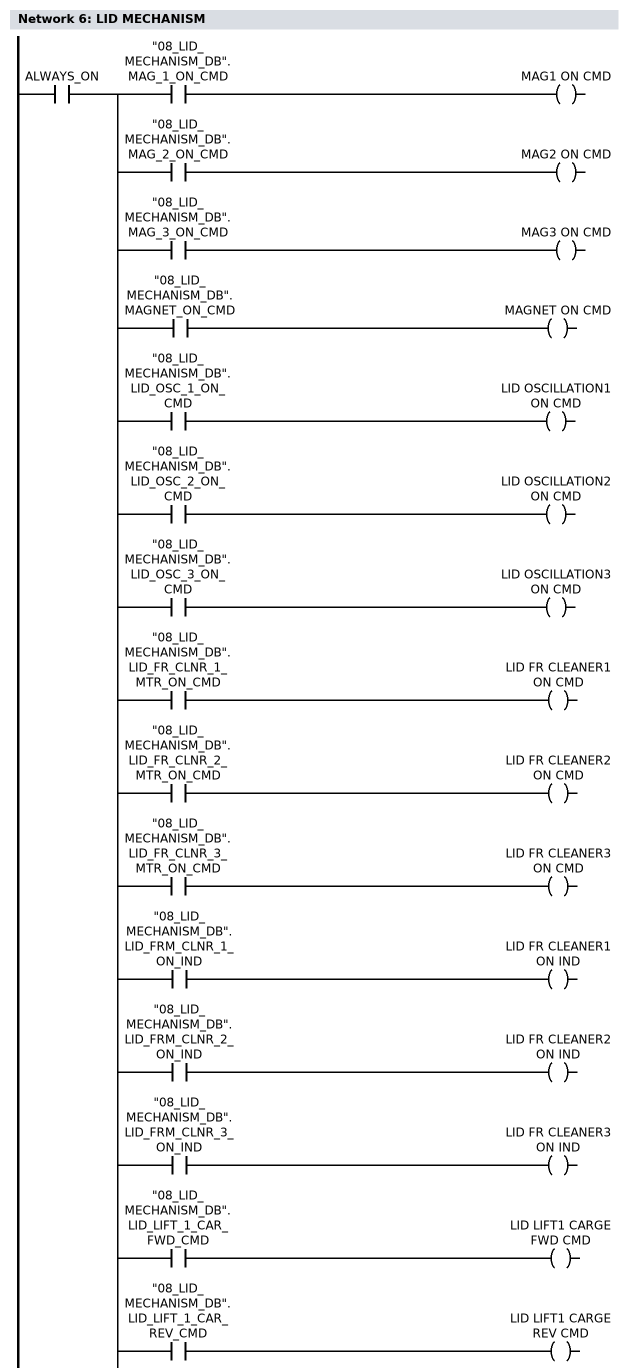
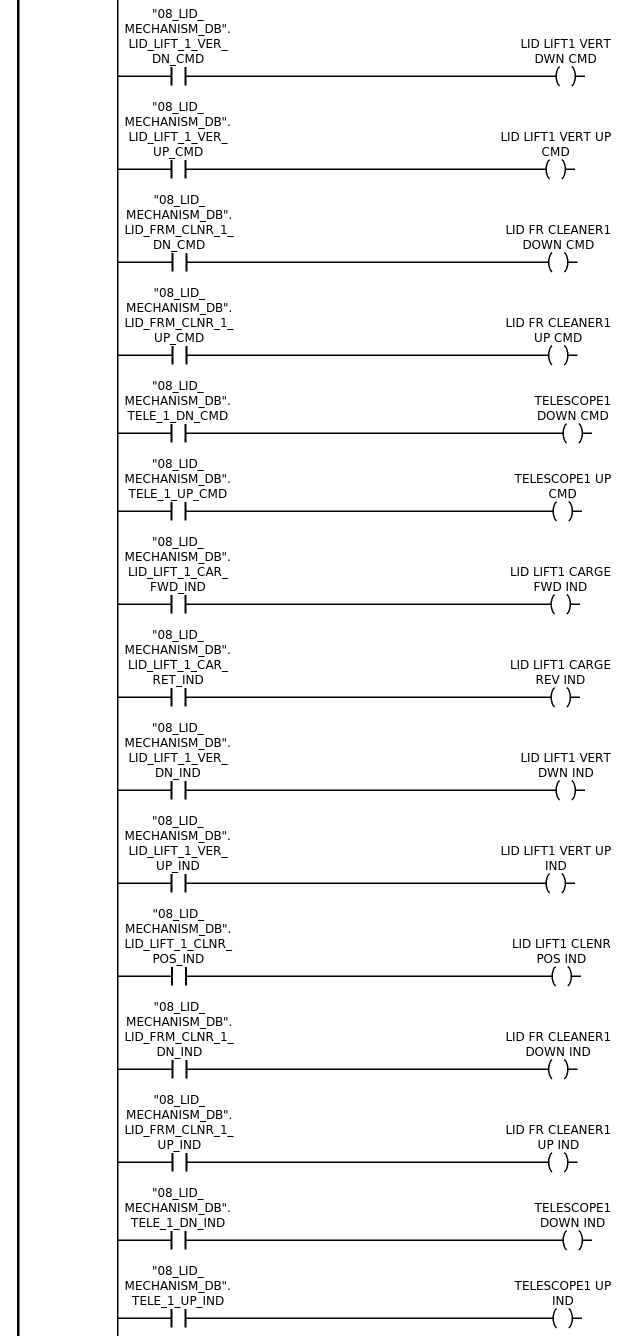
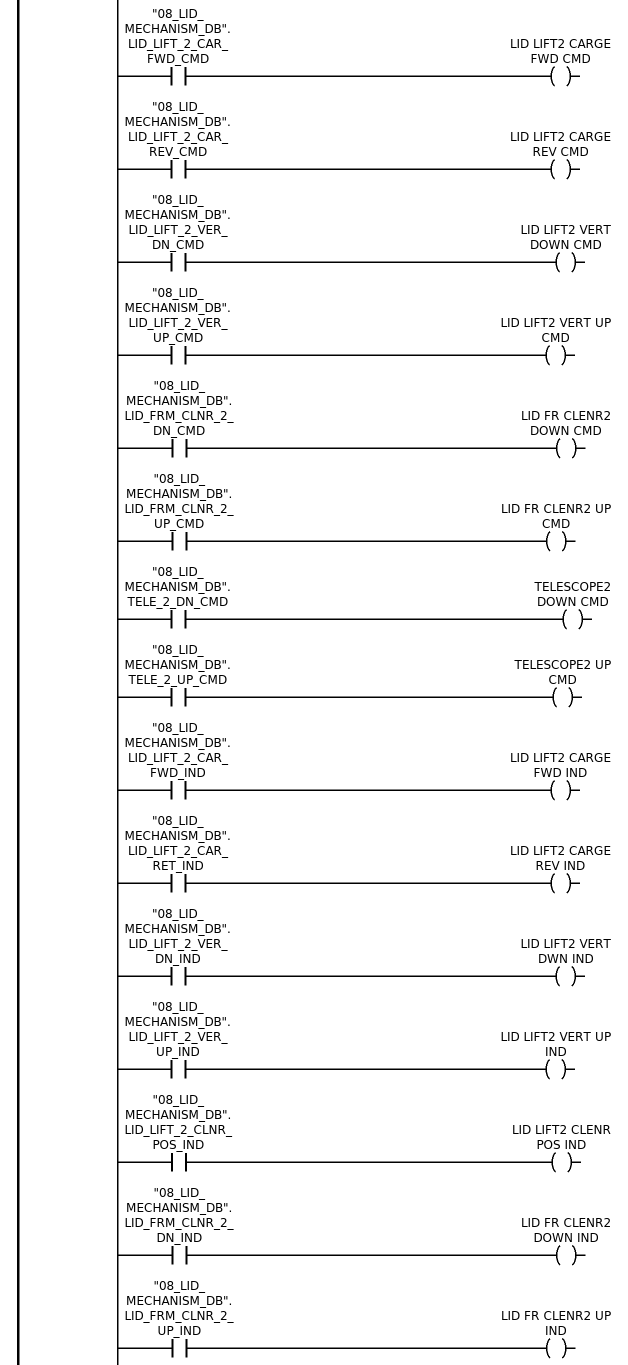
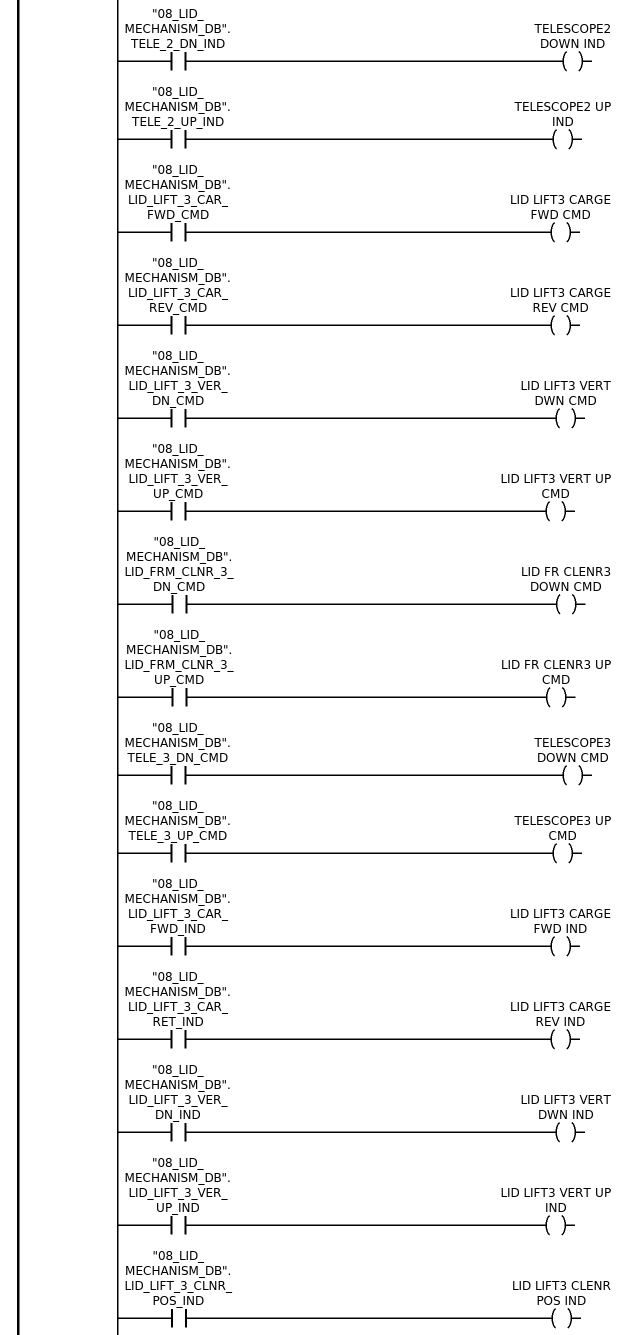
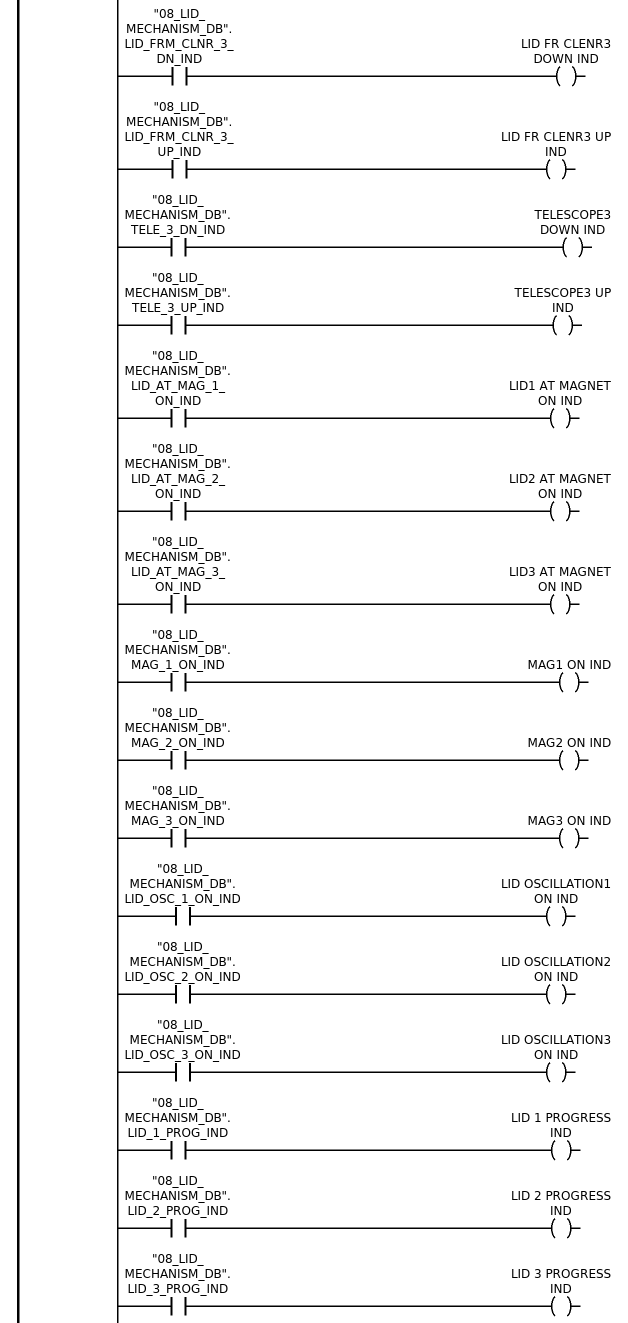
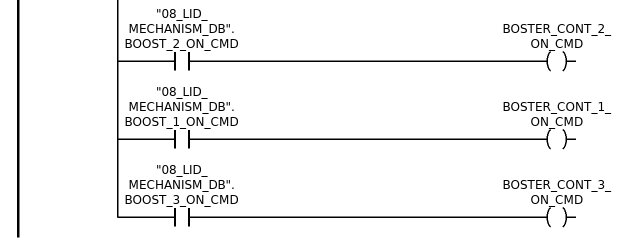
NETWORK
TITLE = LID MECHANISM
      A     "ALWAYS_ON";
      =     L 0.0;
      A     L 0.0;
      A     "08_LID_MECHANISM_DB".MAG_1_ON_CMD;
      =     "MAG1 ON CMD";
      A     L 0.0;
      A     "08_LID_MECHANISM_DB".MAG_2_ON_CMD;
      =     "MAG2 ON CMD";
      A     L 0.0;
      A     "08_LID_MECHANISM_DB".MAG_3_ON_CMD;
      =     "MAG3 ON CMD";
      A     L 0.0;
      A     "08_LID_MECHANISM_DB".MAGNET_ON_CMD;
      =     "MAGNET ON CMD";
      A     L 0.0;
      A     "08_LID_MECHANISM_DB".LID_OSC_1_ON_CMD;
      =     "LID OSCILLATION1 ON CMD";
      A     L 0.0;
      A     "08_LID_MECHANISM_DB".LID_OSC_2_ON_CMD;
      =     "LID OSCILLATION2 ON CMD";
      A     L 0.0;
      A     "08_LID_MECHANISM_DB".LID_OSC_3_ON_CMD;
      =     "LID OSCILLATION3 ON CMD";
      A     L 0.0;
      A     "08_LID_MECHANISM_DB".LID_FR_CLNR_1_MTR_ON_CMD;
      =     "LID FR CLEANER1 ON CMD";
      A     L 0.0;
      A     "08_LID_MECHANISM_DB".LID_FR_CLNR_2_MTR_ON_CMD;
      =     "LID FR CLEANER2 ON CMD";
      A     L 0.0;
      A     "08_LID_MECHANISM_DB".LID_FR_CLNR_3_MTR_ON_CMD;
      =     "LID FR CLEANER3 ON CMD";
      A     L 0.0;
      A     "08_LID_MECHANISM_DB".LID_FRM_CLNR_1_ON_IND;
      =     "LID FR CLEANER1 ON IND";
      A     L 0.0;
      A     "08_LID_MECHANISM_DB".LID_FRM_CLNR_2_ON_IND;
      =     "LID FR CLEANER2 ON IND";
      A     L 0.0;
      A     "08_LID_MECHANISM_DB".LID_FRM_CLNR_3_ON_IND;
      =     "LID FR CLEANER3 ON IND";
      A     L 0.0;
      A     "08_LID_MECHANISM_DB".LID_LIFT_1_CAR_FWD_CMD;
      =     "LID LIFT1 CARGE FWD CMD";
      A     L 0.0;
      A     "08_LID_MECHANISM_DB".LID_LIFT_1_CAR_REV_CMD;
      =     "LID LIFT1 CARGE REV CMD";
      A     L 0.0;
      A     "08_LID_MECHANISM_DB".LID_LIFT_1_VER_DN_CMD;
      =     "LID LIFT1 VERT DWN CMD";
      A     L 0.0;
      A     "08_LID_MECHANISM_DB".LID_LIFT_1_VER_UP_CMD;
      =     "LID LIFT1 VERT UP CMD";
      A     L 0.0;
      A     "08_LID_MECHANISM_DB".LID_FRM_CLNR_1_DN_CMD;
      =     "LID FR CLEANER1 DOWN CMD";
      A     L 0.0;
      A     "08_LID_MECHANISM_DB".LID_FRM_CLNR_1_UP_CMD;
      =     "LID FR CLEANER1 UP CMD";
      A     L 0.0;
      A     "08_LID_MECHANISM_DB".TELE_1_DN_CMD;
      =     "TELESCOPE1 DOWN CMD";
      A     L 0.0;
      A     "08_LID_MECHANISM_DB".TELE_1_UP_CMD;
      =     "TELESCOPE1 UP CMD";
      A     L 0.0;
      A     "08_LID_MECHANISM_DB".LID_LIFT_1_CAR_FWD_IND;
      =     "LID LIFT1 CARGE FWD IND";
      A     L 0.0;
      A     "08_LID_MECHANISM_DB".LID_LIFT_1_CAR_RET_IND;
      =     "LID LIFT1 CARGE REV IND";
      A     L 0.0;
      A     "08_LID_MECHANISM_DB".LID_LIFT_1_VER_DN_IND;
      =     "LID LIFT1 VERT DWN IND";
      A     L 0.0;
      A     "08_LID_MECHANISM_DB".LID_LIFT_1_VER_UP_IND;
      =     "LID LIFT1 VERT UP IND";
      A     L 0.0;
      A     "08_LID_MECHANISM_DB".LID_LIFT_1_CLNR_POS_IND;
      =     "LID LIFT1 CLENR POS IND";
      A     L 0.0;
      A     "08_LID_MECHANISM_DB".LID_FRM_CLNR_1_DN_IND;
      =     "LID FR CLEANER1 DOWN IND";
      A     L 0.0;
      A     "08_LID_MECHANISM_DB".LID_FRM_CLNR_1_UP_IND;
      =     "LID FR CLEANER1 UP IND";
      A     L 0.0;
      A     "08_LID_MECHANISM_DB".TELE_1_DN_IND;
      =     "TELESCOPE1 DOWN IND";
      A     L 0.0;
      A     "08_LID_MECHANISM_DB".TELE_1_UP_IND;
      =     "TELESCOPE1 UP IND";
      A     L 0.0;
      A     "08_LID_MECHANISM_DB".LID_LIFT_2_CAR_FWD_CMD;
      =     "LID LIFT2 CARGE FWD CMD";
      A     L 0.0;
      A     "08_LID_MECHANISM_DB".LID_LIFT_2_CAR_REV_CMD;
      =     "LID LIFT2 CARGE REV CMD";
      A     L 0.0;
      A     "08_LID_MECHANISM_DB".LID_LIFT_2_VER_DN_CMD;
      =     "LID LIFT2 VERT DOWN CMD";
      A     L 0.0;
      A     "08_LID_MECHANISM_DB".LID_LIFT_2_VER_UP_CMD;
      =     "LID LIFT2 VERT UP CMD";
      A     L 0.0;
      A     "08_LID_MECHANISM_DB".LID_FRM_CLNR_2_DN_CMD;
      =     "LID FR CLENR2 DOWN CMD";
      A     L 0.0;
      A     "08_LID_MECHANISM_DB".LID_FRM_CLNR_2_UP_CMD;
      =     "LID FR CLENR2 UP CMD";
      A     L 0.0;
      A     "08_LID_MECHANISM_DB".TELE_2_DN_CMD;
      =     "TELESCOPE2 DOWN CMD";
      A     L 0.0;
      A     "08_LID_MECHANISM_DB".TELE_2_UP_CMD;
      =     "TELESCOPE2 UP CMD";
      A     L 0.0;
      A     "08_LID_MECHANISM_DB".LID_LIFT_2_CAR_FWD_IND;
      =     "LID LIFT2 CARGE FWD IND";
      A     L 0.0;
      A     "08_LID_MECHANISM_DB".LID_LIFT_2_CAR_RET_IND;
      =     "LID LIFT2 CARGE REV IND";
      A     L 0.0;
      A     "08_LID_MECHANISM_DB".LID_LIFT_2_VER_DN_IND;
      =     "LID LIFT2 VERT DWN IND";
      A     L 0.0;
      A     "08_LID_MECHANISM_DB".LID_LIFT_2_VER_UP_IND;
      =     "LID LIFT2 VERT UP IND";
      A     L 0.0;
      A     "08_LID_MECHANISM_DB".LID_LIFT_2_CLNR_POS_IND;
      =     "LID LIFT2 CLENR POS IND";
      A     L 0.0;
      A     "08_LID_MECHANISM_DB".LID_FRM_CLNR_2_DN_IND;
      =     "LID FR CLENR2 DOWN IND";
      A     L 0.0;
      A     "08_LID_MECHANISM_DB".LID_FRM_CLNR_2_UP_IND;
      =     "LID FR CLENR2 UP IND";
      A     L 0.0;
      A     "08_LID_MECHANISM_DB".TELE_2_DN_IND;
      =     "TELESCOPE2 DOWN IND";
      A     L 0.0;
      A     "08_LID_MECHANISM_DB".TELE_2_UP_IND;
      =     "TELESCOPE2 UP IND";
      A     L 0.0;
      A     "08_LID_MECHANISM_DB".LID_LIFT_3_CAR_FWD_CMD;
      =     "LID LIFT3 CARGE FWD CMD";
      A     L 0.0;
      A     "08_LID_MECHANISM_DB".LID_LIFT_3_CAR_REV_CMD;
      =     "LID LIFT3 CARGE REV CMD";
      A     L 0.0;
      A     "08_LID_MECHANISM_DB".LID_LIFT_3_VER_DN_CMD;
      =     "LID LIFT3 VERT DWN CMD";
      A     L 0.0;
      A     "08_LID_MECHANISM_DB".LID_LIFT_3_VER_UP_CMD;
      =     "LID LIFT3 VERT UP CMD";
      A     L 0.0;
      A     "08_LID_MECHANISM_DB".LID_FRM_CLNR_3_DN_CMD;
      =     "LID FR CLENR3 DOWN CMD";
      A     L 0.0;
      A     "08_LID_MECHANISM_DB".LID_FRM_CLNR_3_UP_CMD;
      =     "LID FR CLENR3 UP CMD";
      A     L 0.0;
      A     "08_LID_MECHANISM_DB".TELE_3_DN_CMD;
      =     "TELESCOPE3 DOWN CMD";
      A     L 0.0;
      A     "08_LID_MECHANISM_DB".TELE_3_UP_CMD;
      =     "TELESCOPE3 UP CMD";
      A     L 0.0;
      A     "08_LID_MECHANISM_DB".LID_LIFT_3_CAR_FWD_IND;
      =     "LID LIFT3 CARGE FWD IND";
      A     L 0.0;
      A     "08_LID_MECHANISM_DB".LID_LIFT_3_CAR_RET_IND;
      =     "LID LIFT3 CARGE REV IND";
      A     L 0.0;
      A     "08_LID_MECHANISM_DB".LID_LIFT_3_VER_DN_IND;
      =     "LID LIFT3 VERT DWN IND";
      A     L 0.0;
      A     "08_LID_MECHANISM_DB".LID_LIFT_3_VER_UP_IND;
      =     "LID LIFT3 VERT UP IND";
      A     L 0.0;
      A     "08_LID_MECHANISM_DB".LID_LIFT_3_CLNR_POS_IND;
      =     "LID LIFT3 CLENR POS IND";
      A     L 0.0;
      A     "08_LID_MECHANISM_DB".LID_FRM_CLNR_3_DN_IND;
      =     "LID FR CLENR3 DOWN IND";
      A     L 0.0;
      A     "08_LID_MECHANISM_DB".LID_FRM_CLNR_3_UP_IND;
      =     "LID FR CLENR3 UP IND";
      A     L 0.0;
      A     "08_LID_MECHANISM_DB".TELE_3_DN_IND;
      =     "TELESCOPE3 DOWN IND";
      A     L 0.0;
      A     "08_LID_MECHANISM_DB".TELE_3_UP_IND;
      =     "TELESCOPE3 UP IND";
      A     L 0.0;
      A     "08_LID_MECHANISM_DB".LID_AT_MAG_1_ON_IND;
      =     "LID1 AT MAGNET ON IND";
      A     L 0.0;
      A     "08_LID_MECHANISM_DB".LID_AT_MAG_2_ON_IND;
      =     "LID2 AT MAGNET ON IND";
      A     L 0.0;
      A     "08_LID_MECHANISM_DB".LID_AT_MAG_3_ON_IND;
      =     "LID3 AT MAGNET ON IND";
      A     L 0.0;
      A     "08_LID_MECHANISM_DB".MAG_1_ON_IND;
      =     "MAG1 ON IND";
      A     L 0.0;
      A     "08_LID_MECHANISM_DB".MAG_2_ON_IND;
      =     "MAG2 ON IND";
      A     L 0.0;
      A     "08_LID_MECHANISM_DB".MAG_3_ON_IND;
      =     "MAG3 ON IND";
      A     L 0.0;
      A     "08_LID_MECHANISM_DB".LID_OSC_1_ON_IND;
      =     "LID OSCILLATION1 ON IND";
      A     L 0.0;
      A     "08_LID_MECHANISM_DB".LID_OSC_2_ON_IND;
      =     "LID OSCILLATION2 ON IND";
      A     L 0.0;
      A     "08_LID_MECHANISM_DB".LID_OSC_3_ON_IND;
      =     "LID OSCILLATION3 ON IND";
      A     L 0.0;
      A     "08_LID_MECHANISM_DB".LID_1_PROG_IND;
      =     "LID 1 PROGRESS IND";
      A     L 0.0;
      A     "08_LID_MECHANISM_DB".LID_2_PROG_IND;
      =     "LID 2 PROGRESS IND";
      A     L 0.0;
      A     "08_LID_MECHANISM_DB".LID_3_PROG_IND;
      =     "LID 3 PROGRESS IND";
      A     L 0.0;
      A     "08_LID_MECHANISM_DB".BOOST_2_ON_CMD;
      =     "BOSTER_CONT_2_ON_CMD";
      A     L 0.0;
      A     "08_LID_MECHANISM_DB".BOOST_1_ON_CMD;
      =     "BOSTER_CONT_1_ON_CMD";
      A     L 0.0;
      A     "08_LID_MECHANISM_DB".BOOST_3_ON_CMD;
      =     "BOSTER_CONT_3_ON_CMD";
END_FUNCTION

FUNCTION "HYDRALIC_FUNCTION" : VOID	// FC 7
AUTHOR : Arun_Ram
VERSION : 0.1
BEGIN
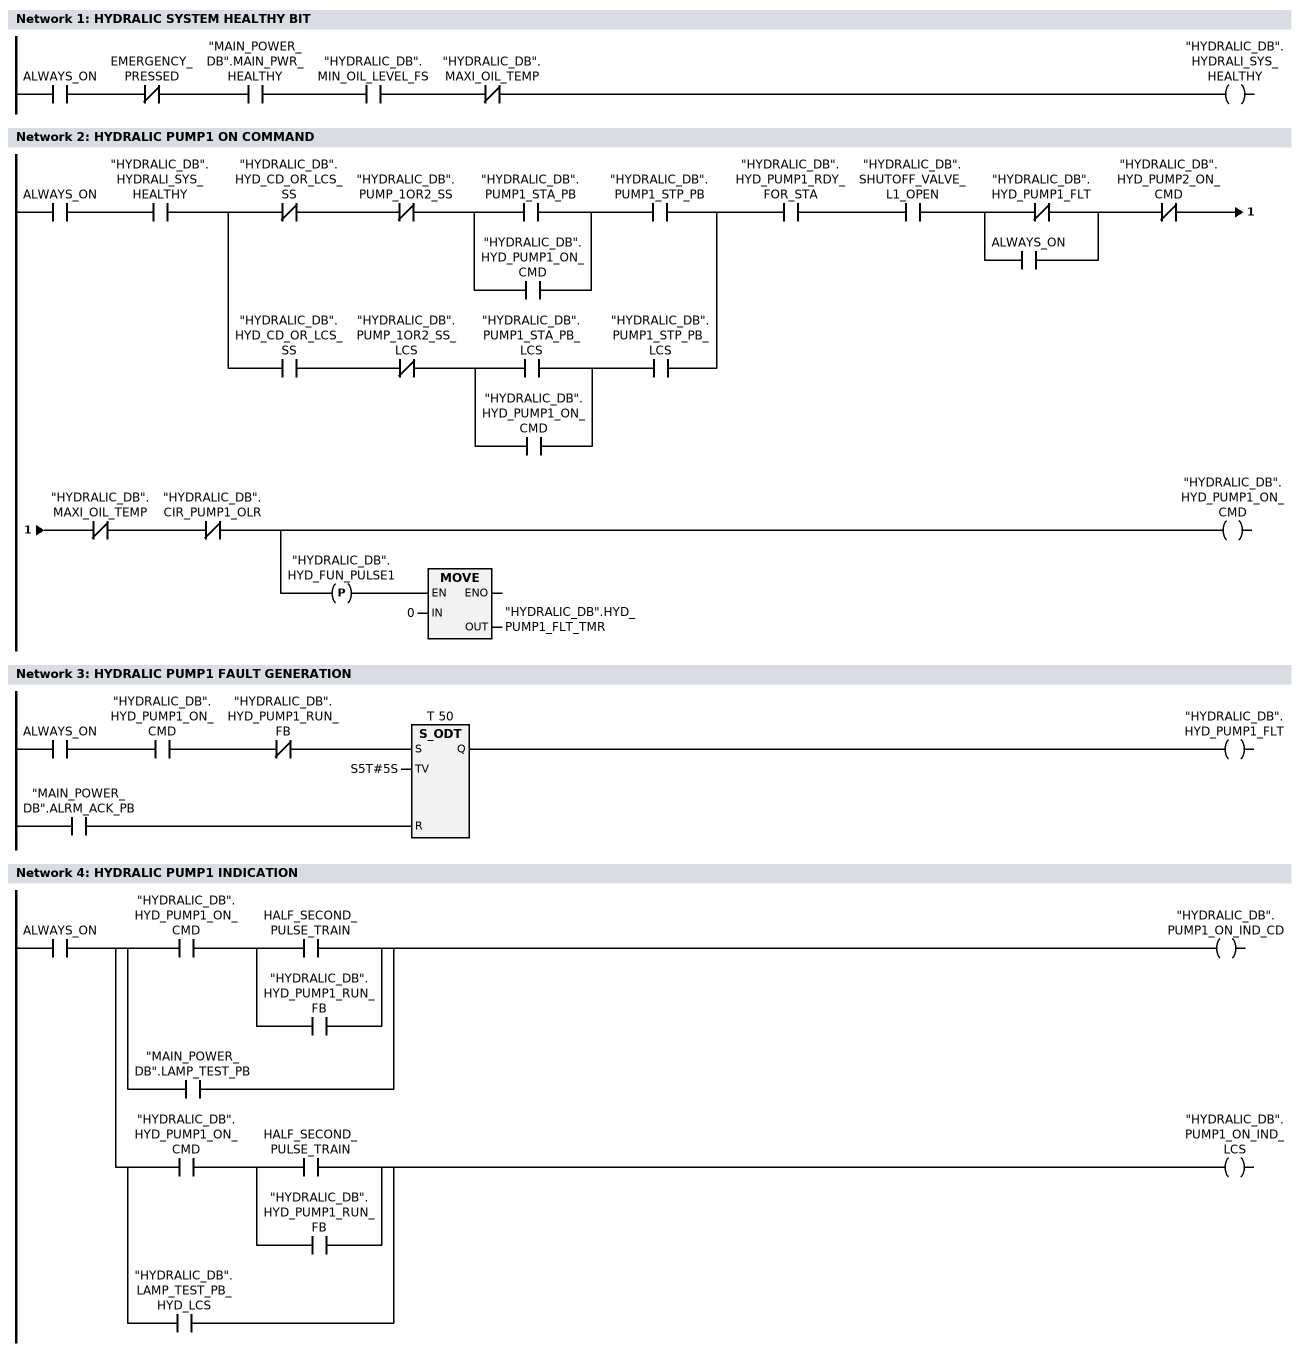
NETWORK
TITLE = HYDRALIC SYSTEM HEALTHY BIT
      A     "ALWAYS_ON";
      AN    "EMERGENCY_PRESSED";
      A     "MAIN_POWER_DB".MAIN_PWR_HEALTHY;
      A     "HYDRALIC_DB".MIN_OIL_LEVEL_FS;
      AN    "HYDRALIC_DB".MAXI_OIL_TEMP;
      =     "HYDRALIC_DB".HYDRALI_SYS_HEALTHY;
NETWORK
TITLE = HYDRALIC PUMP1 ON COMMAND
      A     "ALWAYS_ON";
      A     "HYDRALIC_DB".HYDRALI_SYS_HEALTHY;
      A(;
      AN    "HYDRALIC_DB".HYD_CD_OR_LCS_SS;
      AN    "HYDRALIC_DB".PUMP_1OR2_SS;
      A(;
      O     "HYDRALIC_DB".PUMP1_STA_PB;
      O     "HYDRALIC_DB".HYD_PUMP1_ON_CMD;
      );
      A     "HYDRALIC_DB".PUMP1_STP_PB;
      O;
      A     "HYDRALIC_DB".HYD_CD_OR_LCS_SS;
      AN    "HYDRALIC_DB".PUMP_1OR2_SS_LCS;
      A(;
      O     "HYDRALIC_DB".PUMP1_STA_PB_LCS;
      O     "HYDRALIC_DB".HYD_PUMP1_ON_CMD;
      );
      A     "HYDRALIC_DB".PUMP1_STP_PB_LCS;
      );
      A     "HYDRALIC_DB".HYD_PUMP1_RDY_FOR_STA;
      A     "HYDRALIC_DB".SHUTOFF_VALVE_L1_OPEN;
      A(;
      ON    "HYDRALIC_DB".HYD_PUMP1_FLT;
      O     "ALWAYS_ON";
      );
      AN    "HYDRALIC_DB".HYD_PUMP2_ON_CMD;
      AN    "HYDRALIC_DB".MAXI_OIL_TEMP;
      AN    "HYDRALIC_DB".CIR_PUMP1_OLR;
      =     L 0.0;
      A     L 0.0;
      BLD   102;
      =     "HYDRALIC_DB".HYD_PUMP1_ON_CMD;
      A     L 0.0;
      FP    "HYDRALIC_DB".HYD_FUN_PULSE1;
      JNB   _001;
      L     0;
      T     "HYDRALIC_DB".HYD_PUMP1_FLT_TMR;
_001: NOP   0;
NETWORK
TITLE = HYDRALIC PUMP1 FAULT GENERATION
      A     "ALWAYS_ON";
      A     "HYDRALIC_DB".HYD_PUMP1_ON_CMD;
      AN    "HYDRALIC_DB".HYD_PUMP1_RUN_FB;
      L     S5T#5S;
      SD    T 50;
      A     "MAIN_POWER_DB".ALRM_ACK_PB;
      R     T 50;
      NOP   0;
      NOP   0;
      A     T 50;
      =     "HYDRALIC_DB".HYD_PUMP1_FLT;
NETWORK
TITLE = HYDRALIC PUMP1 INDICATION
      A     "ALWAYS_ON";
      =     L 0.0;
      A     L 0.0;
      A(;
      A     "HYDRALIC_DB".HYD_PUMP1_ON_CMD;
      A(;
      O     "HALF_SECOND_PULSE_TRAIN";
      O     "HYDRALIC_DB".HYD_PUMP1_RUN_FB;
      );
      O     "MAIN_POWER_DB".LAMP_TEST_PB;
      );
      =     "HYDRALIC_DB".PUMP1_ON_IND_CD;
      A     L 0.0;
      A(;
      A     "HYDRALIC_DB".HYD_PUMP1_ON_CMD;
      A(;
      O     "HALF_SECOND_PULSE_TRAIN";
      O     "HYDRALIC_DB".HYD_PUMP1_RUN_FB;
      );
      O     "HYDRALIC_DB".LAMP_TEST_PB_HYD_LCS;
      );
      =     "HYDRALIC_DB".PUMP1_ON_IND_LCS;
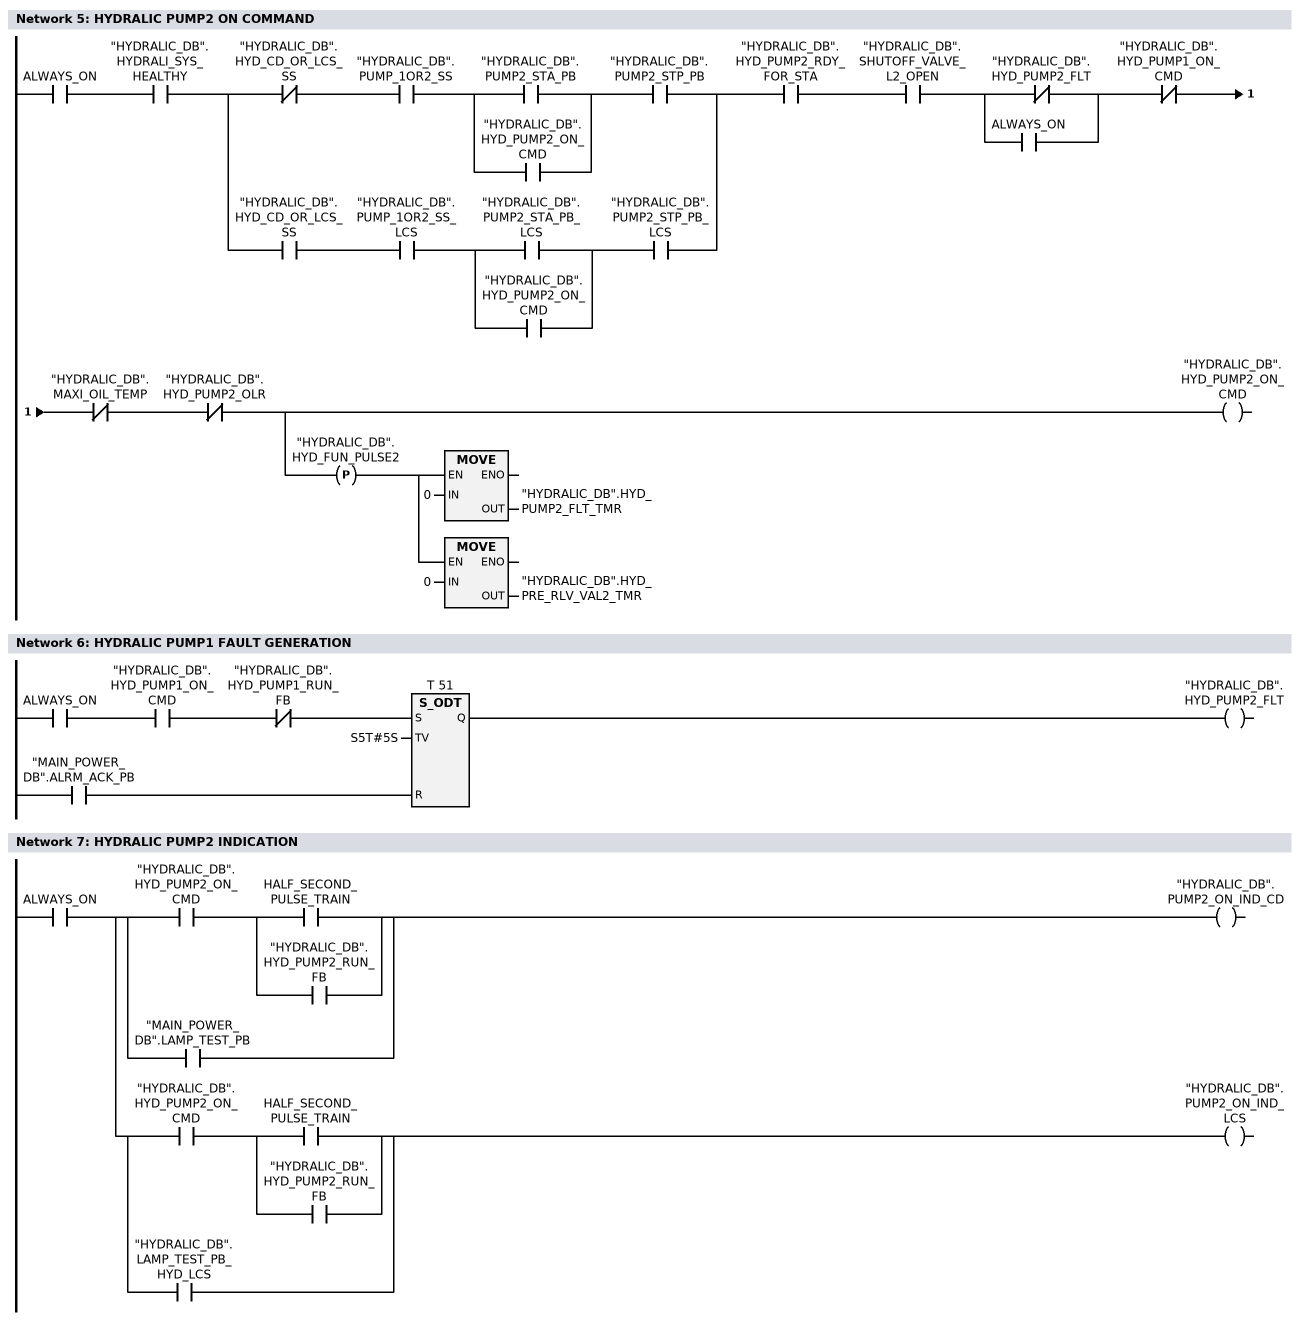
NETWORK
TITLE = HYDRALIC PUMP2 ON COMMAND
      A     "ALWAYS_ON";
      A     "HYDRALIC_DB".HYDRALI_SYS_HEALTHY;
      A(;
      AN    "HYDRALIC_DB".HYD_CD_OR_LCS_SS;
      A     "HYDRALIC_DB".PUMP_1OR2_SS;
      A(;
      O     "HYDRALIC_DB".PUMP2_STA_PB;
      O     "HYDRALIC_DB".HYD_PUMP2_ON_CMD;
      );
      A     "HYDRALIC_DB".PUMP2_STP_PB;
      O;
      A     "HYDRALIC_DB".HYD_CD_OR_LCS_SS;
      A     "HYDRALIC_DB".PUMP_1OR2_SS_LCS;
      A(;
      O     "HYDRALIC_DB".PUMP2_STA_PB_LCS;
      O     "HYDRALIC_DB".HYD_PUMP2_ON_CMD;
      );
      A     "HYDRALIC_DB".PUMP2_STP_PB_LCS;
      );
      A     "HYDRALIC_DB".HYD_PUMP2_RDY_FOR_STA;
      A     "HYDRALIC_DB".SHUTOFF_VALVE_L2_OPEN;
      A(;
      ON    "HYDRALIC_DB".HYD_PUMP2_FLT;
      O     "ALWAYS_ON";
      );
      AN    "HYDRALIC_DB".HYD_PUMP1_ON_CMD;
      AN    "HYDRALIC_DB".MAXI_OIL_TEMP;
      AN    "HYDRALIC_DB".HYD_PUMP2_OLR;
      =     L 0.0;
      A     L 0.0;
      BLD   102;
      =     "HYDRALIC_DB".HYD_PUMP2_ON_CMD;
      A     L 0.0;
      FP    "HYDRALIC_DB".HYD_FUN_PULSE2;
      =     L 0.1;
      A     L 0.1;
      JNB   _002;
      L     0;
      T     "HYDRALIC_DB".HYD_PUMP2_FLT_TMR;
_002: NOP   0;
      A     L 0.1;
      JNB   _003;
      L     0;
      T     "HYDRALIC_DB".HYD_PRE_RLV_VAL2_TMR;
_003: NOP   0;
NETWORK
TITLE = HYDRALIC PUMP1 FAULT GENERATION
      A     "ALWAYS_ON";
      A     "HYDRALIC_DB".HYD_PUMP1_ON_CMD;
      AN    "HYDRALIC_DB".HYD_PUMP1_RUN_FB;
      L     S5T#5S;
      SD    T 51;
      A     "MAIN_POWER_DB".ALRM_ACK_PB;
      R     T 51;
      NOP   0;
      NOP   0;
      A     T 51;
      =     "HYDRALIC_DB".HYD_PUMP2_FLT;
NETWORK
TITLE = HYDRALIC PUMP2 INDICATION
      A     "ALWAYS_ON";
      =     L 0.0;
      A     L 0.0;
      A(;
      A     "HYDRALIC_DB".HYD_PUMP2_ON_CMD;
      A(;
      O     "HALF_SECOND_PULSE_TRAIN";
      O     "HYDRALIC_DB".HYD_PUMP2_RUN_FB;
      );
      O     "MAIN_POWER_DB".LAMP_TEST_PB;
      );
      =     "HYDRALIC_DB".PUMP2_ON_IND_CD;
      A     L 0.0;
      A(;
      A     "HYDRALIC_DB".HYD_PUMP2_ON_CMD;
      A(;
      O     "HALF_SECOND_PULSE_TRAIN";
      O     "HYDRALIC_DB".HYD_PUMP2_RUN_FB;
      );
      O     "HYDRALIC_DB".LAMP_TEST_PB_HYD_LCS;
      );
      =     "HYDRALIC_DB".PUMP2_ON_IND_LCS;
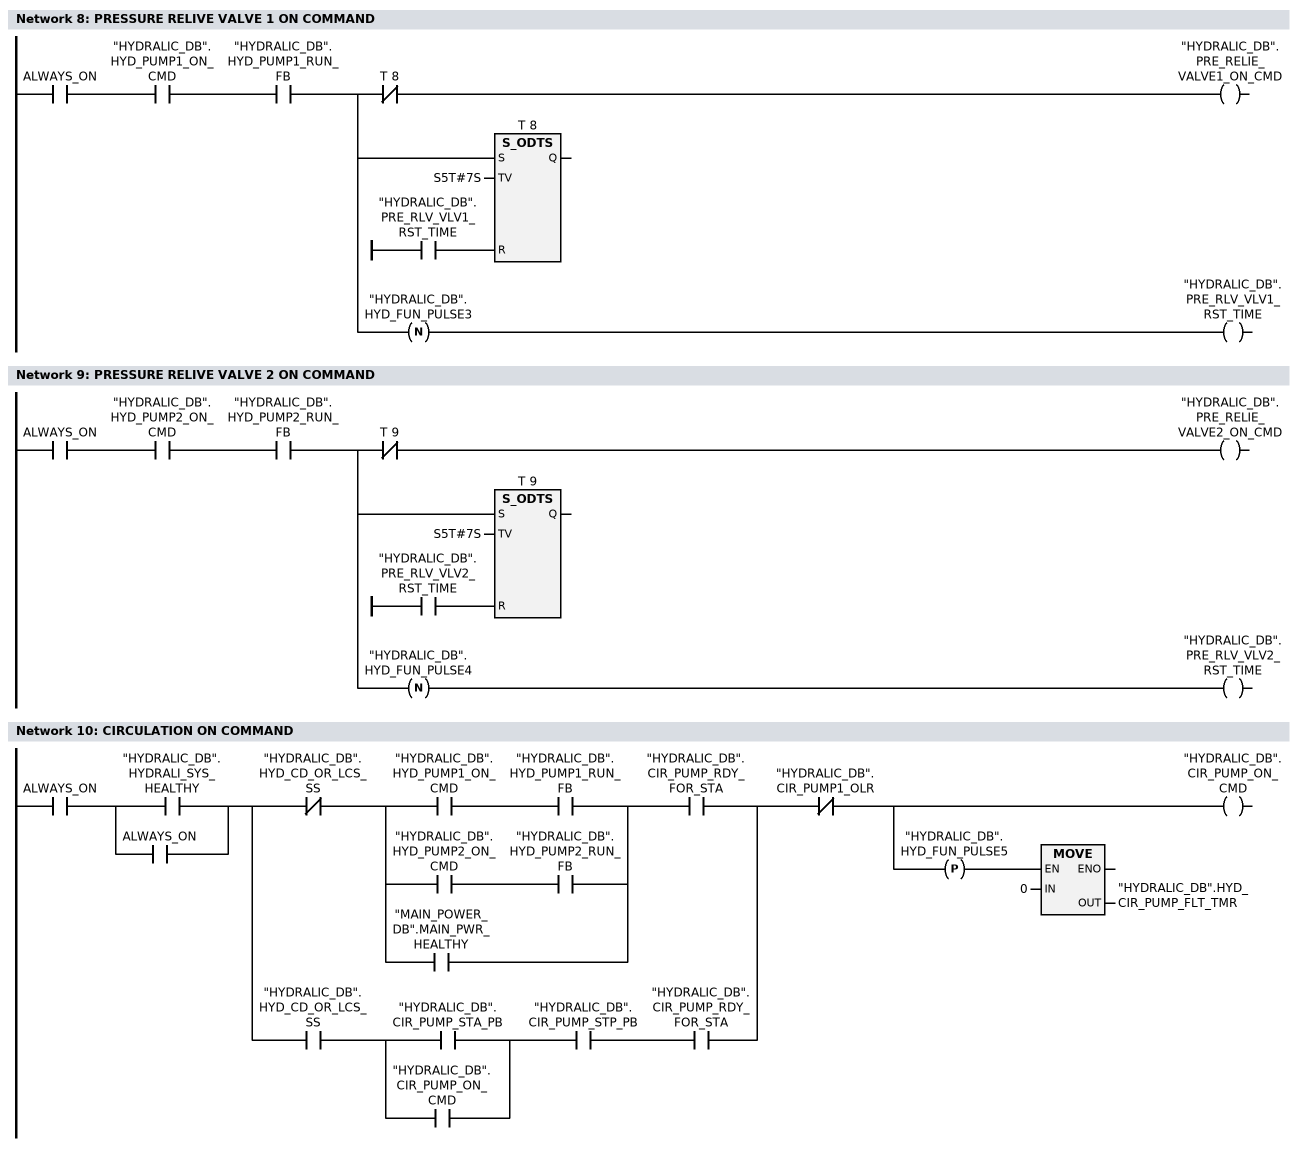
NETWORK
TITLE = PRESSURE RELIVE VALVE 1 ON COMMAND
      A     "ALWAYS_ON";
      A     "HYDRALIC_DB".HYD_PUMP1_ON_CMD;
      A     "HYDRALIC_DB".HYD_PUMP1_RUN_FB;
      =     L 0.0;
      A     L 0.0;
      AN    T 8;
      =     "HYDRALIC_DB".PRE_RELIE_VALVE1_ON_CMD;
      A     L 0.0;
      L     S5T#7S;
      SS    T 8;
      A     "HYDRALIC_DB".PRE_RLV_VLV1_RST_TIME;
      R     T 8;
      NOP   0;
      NOP   0;
      NOP   0;
      A     L 0.0;
      FN    "HYDRALIC_DB".HYD_FUN_PULSE3;
      =     "HYDRALIC_DB".PRE_RLV_VLV1_RST_TIME;
NETWORK
TITLE = PRESSURE RELIVE VALVE 2 ON COMMAND
      A     "ALWAYS_ON";
      A     "HYDRALIC_DB".HYD_PUMP2_ON_CMD;
      A     "HYDRALIC_DB".HYD_PUMP2_RUN_FB;
      =     L 0.0;
      A     L 0.0;
      AN    T 9;
      =     "HYDRALIC_DB".PRE_RELIE_VALVE2_ON_CMD;
      A     L 0.0;
      L     S5T#7S;
      SS    T 9;
      A     "HYDRALIC_DB".PRE_RLV_VLV2_RST_TIME;
      R     T 9;
      NOP   0;
      NOP   0;
      NOP   0;
      A     L 0.0;
      FN    "HYDRALIC_DB".HYD_FUN_PULSE4;
      =     "HYDRALIC_DB".PRE_RLV_VLV2_RST_TIME;
NETWORK
TITLE = CIRCULATION ON COMMAND
      A     "ALWAYS_ON";
      A(;
      O     "HYDRALIC_DB".HYDRALI_SYS_HEALTHY;
      O     "ALWAYS_ON";
      );
      A(;
      AN    "HYDRALIC_DB".HYD_CD_OR_LCS_SS;
      A(;
      A     "HYDRALIC_DB".HYD_PUMP1_ON_CMD;
      A     "HYDRALIC_DB".HYD_PUMP1_RUN_FB;
      O;
      A     "HYDRALIC_DB".HYD_PUMP2_ON_CMD;
      A     "HYDRALIC_DB".HYD_PUMP2_RUN_FB;
      O     "MAIN_POWER_DB".MAIN_PWR_HEALTHY;
      );
      A     "HYDRALIC_DB".CIR_PUMP_RDY_FOR_STA;
      O;
      A     "HYDRALIC_DB".HYD_CD_OR_LCS_SS;
      A(;
      O     "HYDRALIC_DB".CIR_PUMP_STA_PB;
      O     "HYDRALIC_DB".CIR_PUMP_ON_CMD;
      );
      A     "HYDRALIC_DB".CIR_PUMP_STP_PB;
      A     "HYDRALIC_DB".CIR_PUMP_RDY_FOR_STA;
      );
      AN    "HYDRALIC_DB".CIR_PUMP1_OLR;
      =     L 0.0;
      A     L 0.0;
      BLD   102;
      =     "HYDRALIC_DB".CIR_PUMP_ON_CMD;
      A     L 0.0;
      FP    "HYDRALIC_DB".HYD_FUN_PULSE5;
      JNB   _004;
      L     0;
      T     "HYDRALIC_DB".HYD_CIR_PUMP_FLT_TMR;
_004: NOP   0;
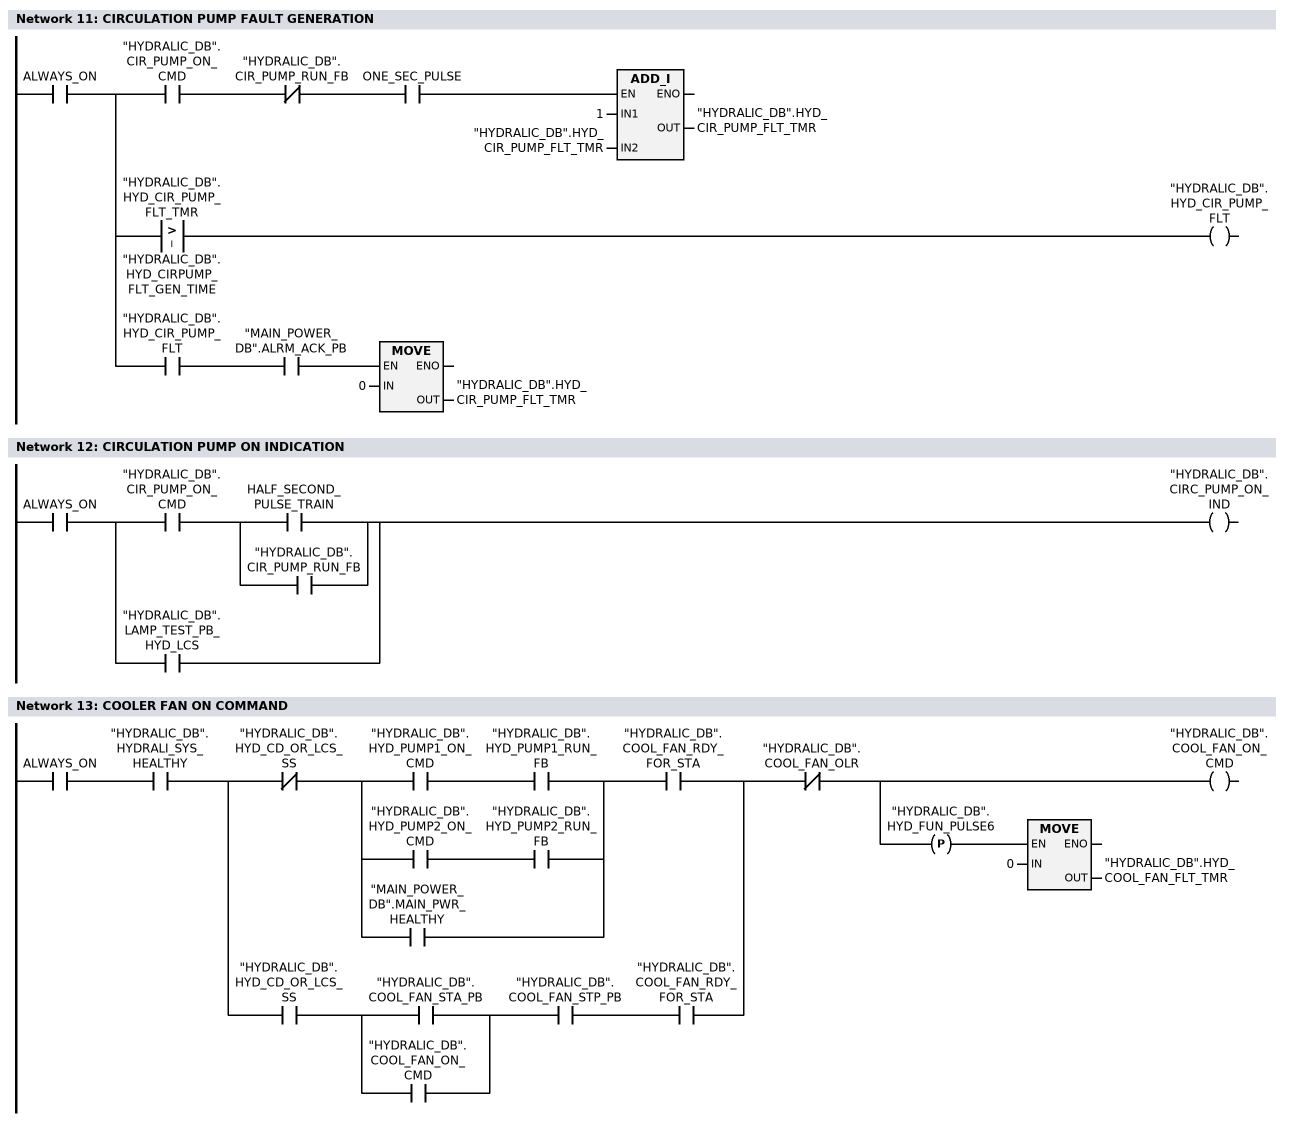
NETWORK
TITLE = CIRCULATION PUMP FAULT GENERATION
      A     "ALWAYS_ON";
      =     L 0.0;
      A     L 0.0;
      A     "HYDRALIC_DB".CIR_PUMP_ON_CMD;
      AN    "HYDRALIC_DB".CIR_PUMP_RUN_FB;
      A     "ONE_SEC_PULSE";
      JNB   _005;
      L     1;
      L     "HYDRALIC_DB".HYD_CIR_PUMP_FLT_TMR;
      +I;
      T     "HYDRALIC_DB".HYD_CIR_PUMP_FLT_TMR;
_005: NOP   0;
      A     L 0.0;
      A(;
      L     "HYDRALIC_DB".HYD_CIR_PUMP_FLT_TMR;
      L     "HYDRALIC_DB".HYD_CIRPUMP_FLT_GEN_TIME;
      >I;
      );
      =     "HYDRALIC_DB".HYD_CIR_PUMP_FLT;
      A     L 0.0;
      A     "HYDRALIC_DB".HYD_CIR_PUMP_FLT;
      A     "MAIN_POWER_DB".ALRM_ACK_PB;
      JNB   _006;
      L     0;
      T     "HYDRALIC_DB".HYD_CIR_PUMP_FLT_TMR;
_006: NOP   0;
NETWORK
TITLE = CIRCULATION PUMP ON INDICATION
      A     "ALWAYS_ON";
      A(;
      A     "HYDRALIC_DB".CIR_PUMP_ON_CMD;
      A(;
      O     "HALF_SECOND_PULSE_TRAIN";
      O     "HYDRALIC_DB".CIR_PUMP_RUN_FB;
      );
      O     "HYDRALIC_DB".LAMP_TEST_PB_HYD_LCS;
      );
      =     "HYDRALIC_DB".CIRC_PUMP_ON_IND;
NETWORK
TITLE = COOLER FAN ON COMMAND
      A     "ALWAYS_ON";
      A     "HYDRALIC_DB".HYDRALI_SYS_HEALTHY;
      A(;
      AN    "HYDRALIC_DB".HYD_CD_OR_LCS_SS;
      A(;
      A     "HYDRALIC_DB".HYD_PUMP1_ON_CMD;
      A     "HYDRALIC_DB".HYD_PUMP1_RUN_FB;
      O;
      A     "HYDRALIC_DB".HYD_PUMP2_ON_CMD;
      A     "HYDRALIC_DB".HYD_PUMP2_RUN_FB;
      O     "MAIN_POWER_DB".MAIN_PWR_HEALTHY;
      );
      A     "HYDRALIC_DB".COOL_FAN_RDY_FOR_STA;
      O;
      A     "HYDRALIC_DB".HYD_CD_OR_LCS_SS;
      A(;
      O     "HYDRALIC_DB".COOL_FAN_STA_PB;
      O     "HYDRALIC_DB".COOL_FAN_ON_CMD;
      );
      A     "HYDRALIC_DB".COOL_FAN_STP_PB;
      A     "HYDRALIC_DB".COOL_FAN_RDY_FOR_STA;
      );
      AN    "HYDRALIC_DB".COOL_FAN_OLR;
      =     L 0.0;
      A     L 0.0;
      BLD   102;
      =     "HYDRALIC_DB".COOL_FAN_ON_CMD;
      A     L 0.0;
      FP    "HYDRALIC_DB".HYD_FUN_PULSE6;
      JNB   _007;
      L     0;
      T     "HYDRALIC_DB".HYD_COOL_FAN_FLT_TMR;
_007: NOP   0;
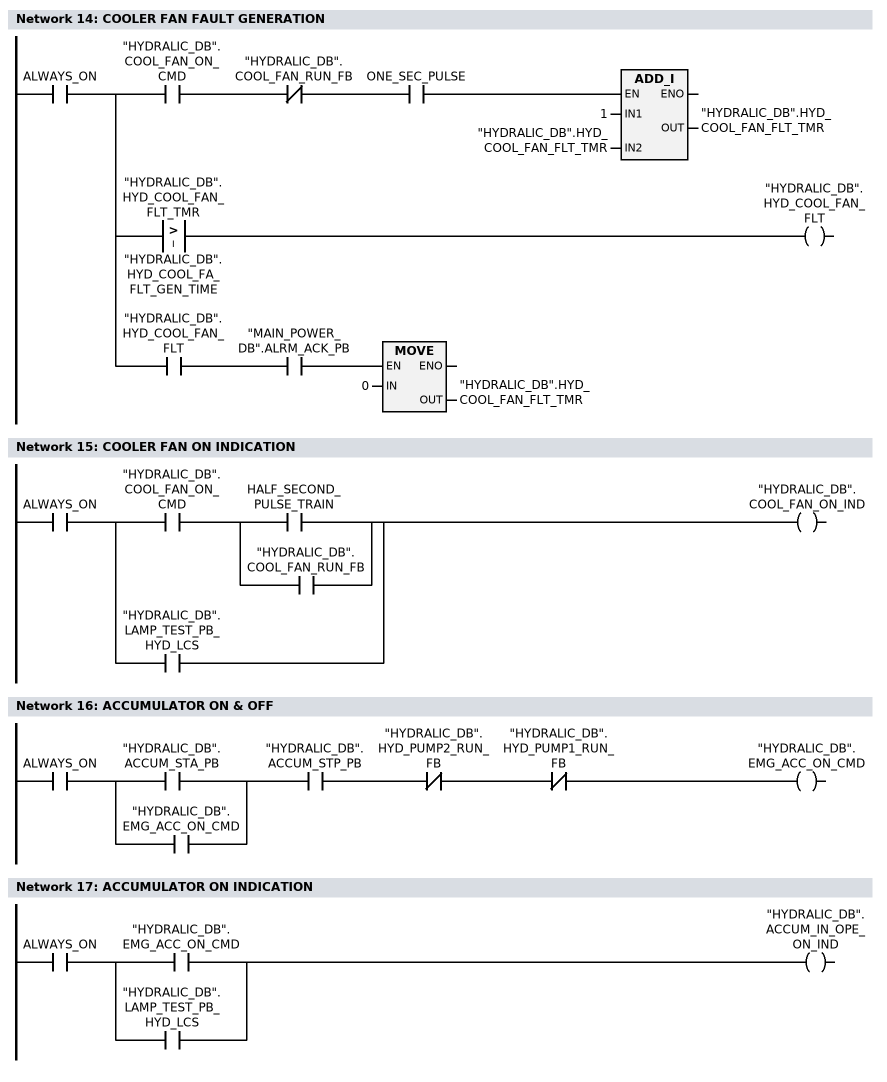
NETWORK
TITLE = COOLER FAN FAULT GENERATION
      A     "ALWAYS_ON";
      =     L 0.0;
      A     L 0.0;
      A     "HYDRALIC_DB".COOL_FAN_ON_CMD;
      AN    "HYDRALIC_DB".COOL_FAN_RUN_FB;
      A     "ONE_SEC_PULSE";
      JNB   _008;
      L     1;
      L     "HYDRALIC_DB".HYD_COOL_FAN_FLT_TMR;
      +I;
      T     "HYDRALIC_DB".HYD_COOL_FAN_FLT_TMR;
_008: NOP   0;
      A     L 0.0;
      A(;
      L     "HYDRALIC_DB".HYD_COOL_FAN_FLT_TMR;
      L     "HYDRALIC_DB".HYD_COOL_FA_FLT_GEN_TIME;
      >I;
      );
      =     "HYDRALIC_DB".HYD_COOL_FAN_FLT;
      A     L 0.0;
      A     "HYDRALIC_DB".HYD_COOL_FAN_FLT;
      A     "MAIN_POWER_DB".ALRM_ACK_PB;
      JNB   _009;
      L     0;
      T     "HYDRALIC_DB".HYD_COOL_FAN_FLT_TMR;
_009: NOP   0;
NETWORK
TITLE = COOLER FAN ON INDICATION
      A     "ALWAYS_ON";
      A(;
      A     "HYDRALIC_DB".COOL_FAN_ON_CMD;
      A(;
      O     "HALF_SECOND_PULSE_TRAIN";
      O     "HYDRALIC_DB".COOL_FAN_RUN_FB;
      );
      O     "HYDRALIC_DB".LAMP_TEST_PB_HYD_LCS;
      );
      =     "HYDRALIC_DB".COOL_FAN_ON_IND;
NETWORK
TITLE = ACCUMULATOR ON & OFF
      A     "ALWAYS_ON";
      A(;
      O     "HYDRALIC_DB".ACCUM_STA_PB;
      O     "HYDRALIC_DB".EMG_ACC_ON_CMD;
      );
      A     "HYDRALIC_DB".ACCUM_STP_PB;
      AN    "HYDRALIC_DB".HYD_PUMP2_RUN_FB;
      AN    "HYDRALIC_DB".HYD_PUMP1_RUN_FB;
      =     "HYDRALIC_DB".EMG_ACC_ON_CMD;
NETWORK
TITLE = ACCUMULATOR ON INDICATION
      A     "ALWAYS_ON";
      A(;
      O     "HYDRALIC_DB".EMG_ACC_ON_CMD;
      O     "HYDRALIC_DB".LAMP_TEST_PB_HYD_LCS;
      );
      =     "HYDRALIC_DB".ACCUM_IN_OPE_ON_IND;
